    stLENS1_750[0].fEnergy := 5960.000000; stLENS1_750[0].fLow := 85.385702; stLENS1_750[0].fHigh := 10000.000000; 
    stLENS1_750[1].fEnergy := 5972.689818; stLENS1_750[1].fLow := 85.043271; stLENS1_750[1].fHigh := 10000.000000; 
    stLENS1_750[2].fEnergy := 5984.647151; stLENS1_750[2].fLow := 84.702213; stLENS1_750[2].fHigh := 10000.000000; 
    stLENS1_750[3].fEnergy := 5996.628422; stLENS1_750[3].fLow := 84.362523; stLENS1_750[3].fHigh := 10000.000000; 
    stLENS1_750[4].fEnergy := 6008.633680; stLENS1_750[4].fLow := 84.024196; stLENS1_750[4].fHigh := 10000.000000; 
    stLENS1_750[5].fEnergy := 6020.662973; stLENS1_750[5].fLow := 83.687225; stLENS1_750[5].fHigh := 10000.000000; 
    stLENS1_750[6].fEnergy := 6032.716348; stLENS1_750[6].fLow := 83.351606; stLENS1_750[6].fHigh := 10000.000000; 
    stLENS1_750[7].fEnergy := 6044.793854; stLENS1_750[7].fLow := 83.017332; stLENS1_750[7].fHigh := 10000.000000; 
    stLENS1_750[8].fEnergy := 6056.895540; stLENS1_750[8].fLow := 82.684399; stLENS1_750[8].fHigh := 10000.000000; 
    stLENS1_750[9].fEnergy := 6069.021453; stLENS1_750[9].fLow := 82.352801; stLENS1_750[9].fHigh := 10000.000000; 
    stLENS1_750[10].fEnergy := 6081.171642; stLENS1_750[10].fLow := 82.022534; stLENS1_750[10].fHigh := 10000.000000; 
    stLENS1_750[11].fEnergy := 6093.346156; stLENS1_750[11].fLow := 81.693590; stLENS1_750[11].fHigh := 10000.000000; 
    stLENS1_750[12].fEnergy := 6105.545043; stLENS1_750[12].fLow := 81.365966; stLENS1_750[12].fHigh := 10000.000000; 
    stLENS1_750[13].fEnergy := 6117.768352; stLENS1_750[13].fLow := 81.039656; stLENS1_750[13].fHigh := 10000.000000; 
    stLENS1_750[14].fEnergy := 6130.016132; stLENS1_750[14].fLow := 80.714654; stLENS1_750[14].fHigh := 10000.000000; 
    stLENS1_750[15].fEnergy := 6142.288433; stLENS1_750[15].fLow := 80.390956; stLENS1_750[15].fHigh := 10000.000000; 
    stLENS1_750[16].fEnergy := 6154.585303; stLENS1_750[16].fLow := 80.068556; stLENS1_750[16].fHigh := 10000.000000; 
    stLENS1_750[17].fEnergy := 6166.906791; stLENS1_750[17].fLow := 79.747449; stLENS1_750[17].fHigh := 10000.000000; 
    stLENS1_750[18].fEnergy := 6179.252946; stLENS1_750[18].fLow := 79.427629; stLENS1_750[18].fHigh := 10000.000000; 
    stLENS1_750[19].fEnergy := 6191.623819; stLENS1_750[19].fLow := 79.109092; stLENS1_750[19].fHigh := 10000.000000; 
    stLENS1_750[20].fEnergy := 6204.019458; stLENS1_750[20].fLow := 78.791833; stLENS1_750[20].fHigh := 10000.000000; 
    stLENS1_750[21].fEnergy := 6216.439913; stLENS1_750[21].fLow := 78.475846; stLENS1_750[21].fHigh := 10000.000000; 
    stLENS1_750[22].fEnergy := 6228.885234; stLENS1_750[22].fLow := 78.161127; stLENS1_750[22].fHigh := 10000.000000; 
    stLENS1_750[23].fEnergy := 6241.355471; stLENS1_750[23].fLow := 77.847669; stLENS1_750[23].fHigh := 10000.000000; 
    stLENS1_750[24].fEnergy := 6253.850673; stLENS1_750[24].fLow := 77.535468; stLENS1_750[24].fHigh := 10000.000000; 
    stLENS1_750[25].fEnergy := 6266.370890; stLENS1_750[25].fLow := 77.224520; stLENS1_750[25].fHigh := 10000.000000; 
    stLENS1_750[26].fEnergy := 6278.916173; stLENS1_750[26].fLow := 76.914819; stLENS1_750[26].fHigh := 10000.000000; 
    stLENS1_750[27].fEnergy := 6291.486572; stLENS1_750[27].fLow := 76.606359; stLENS1_750[27].fHigh := 10000.000000; 
    stLENS1_750[28].fEnergy := 6304.082136; stLENS1_750[28].fLow := 76.299137; stLENS1_750[28].fHigh := 10000.000000; 
    stLENS1_750[29].fEnergy := 6316.702917; stLENS1_750[29].fLow := 75.993147; stLENS1_750[29].fHigh := 10000.000000; 
    stLENS1_750[30].fEnergy := 6329.348965; stLENS1_750[30].fLow := 75.688384; stLENS1_750[30].fHigh := 10000.000000; 
    stLENS1_750[31].fEnergy := 6342.020330; stLENS1_750[31].fLow := 75.384843; stLENS1_750[31].fHigh := 10000.000000; 
    stLENS1_750[32].fEnergy := 6354.717063; stLENS1_750[32].fLow := 75.082519; stLENS1_750[32].fHigh := 10000.000000; 
    stLENS1_750[33].fEnergy := 6367.439215; stLENS1_750[33].fLow := 74.781408; stLENS1_750[33].fHigh := 10000.000000; 
    stLENS1_750[34].fEnergy := 6380.186837; stLENS1_750[34].fLow := 74.481504; stLENS1_750[34].fHigh := 10000.000000; 
    stLENS1_750[35].fEnergy := 6392.959979; stLENS1_750[35].fLow := 74.182804; stLENS1_750[35].fHigh := 10000.000000; 
    stLENS1_750[36].fEnergy := 6405.758694; stLENS1_750[36].fLow := 73.885301; stLENS1_750[36].fHigh := 10000.000000; 
    stLENS1_750[37].fEnergy := 6418.583031; stLENS1_750[37].fLow := 73.588991; stLENS1_750[37].fHigh := 10000.000000; 
    stLENS1_750[38].fEnergy := 6431.433043; stLENS1_750[38].fLow := 73.293869; stLENS1_750[38].fHigh := 10000.000000; 
    stLENS1_750[39].fEnergy := 6444.308780; stLENS1_750[39].fLow := 72.999932; stLENS1_750[39].fHigh := 10000.000000; 
    stLENS1_750[40].fEnergy := 6457.210295; stLENS1_750[40].fLow := 72.707172; stLENS1_750[40].fHigh := 10000.000000; 
    stLENS1_750[41].fEnergy := 6470.137639; stLENS1_750[41].fLow := 72.415587; stLENS1_750[41].fHigh := 10000.000000; 
    stLENS1_750[42].fEnergy := 6483.090863; stLENS1_750[42].fLow := 72.125172; stLENS1_750[42].fHigh := 10000.000000; 
    stLENS1_750[43].fEnergy := 6496.070019; stLENS1_750[43].fLow := 71.835921; stLENS1_750[43].fHigh := 10000.000000; 
    stLENS1_750[44].fEnergy := 6509.075160; stLENS1_750[44].fLow := 71.547830; stLENS1_750[44].fHigh := 10000.000000; 
    stLENS1_750[45].fEnergy := 6522.106337; stLENS1_750[45].fLow := 71.260894; stLENS1_750[45].fHigh := 10000.000000; 
    stLENS1_750[46].fEnergy := 6535.163603; stLENS1_750[46].fLow := 70.975109; stLENS1_750[46].fHigh := 10000.000000; 
    stLENS1_750[47].fEnergy := 6548.247009; stLENS1_750[47].fLow := 70.690471; stLENS1_750[47].fHigh := 10000.000000; 
    stLENS1_750[48].fEnergy := 6561.356609; stLENS1_750[48].fLow := 70.406973; stLENS1_750[48].fHigh := 10000.000000; 
    stLENS1_750[49].fEnergy := 6574.492453; stLENS1_750[49].fLow := 70.124613; stLENS1_750[49].fHigh := 10000.000000; 
    stLENS1_750[50].fEnergy := 6587.654596; stLENS1_750[50].fLow := 69.843385; stLENS1_750[50].fHigh := 10000.000000; 
    stLENS1_750[51].fEnergy := 6600.843089; stLENS1_750[51].fLow := 69.563285; stLENS1_750[51].fHigh := 10000.000000; 
    stLENS1_750[52].fEnergy := 6614.057986; stLENS1_750[52].fLow := 69.284308; stLENS1_750[52].fHigh := 10000.000000; 
    stLENS1_750[53].fEnergy := 6627.299339; stLENS1_750[53].fLow := 69.006450; stLENS1_750[53].fHigh := 10000.000000; 
    stLENS1_750[54].fEnergy := 6640.567201; stLENS1_750[54].fLow := 68.729707; stLENS1_750[54].fHigh := 10000.000000; 
    stLENS1_750[55].fEnergy := 6653.861625; stLENS1_750[55].fLow := 68.454073; stLENS1_750[55].fHigh := 10000.000000; 
    stLENS1_750[56].fEnergy := 6667.182665; stLENS1_750[56].fLow := 68.179545; stLENS1_750[56].fHigh := 10000.000000; 
    stLENS1_750[57].fEnergy := 6680.530374; stLENS1_750[57].fLow := 67.906117; stLENS1_750[57].fHigh := 10000.000000; 
    stLENS1_750[58].fEnergy := 6693.904804; stLENS1_750[58].fLow := 67.633786; stLENS1_750[58].fHigh := 10000.000000; 
    stLENS1_750[59].fEnergy := 6707.306011; stLENS1_750[59].fLow := 67.362548; stLENS1_750[59].fHigh := 10000.000000; 
    stLENS1_750[60].fEnergy := 6720.734046; stLENS1_750[60].fLow := 67.092397; stLENS1_750[60].fHigh := 10000.000000; 
    stLENS1_750[61].fEnergy := 6734.188965; stLENS1_750[61].fLow := 66.823329; stLENS1_750[61].fHigh := 10000.000000; 
    stLENS1_750[62].fEnergy := 6747.670820; stLENS1_750[62].fLow := 66.555341; stLENS1_750[62].fHigh := 10000.000000; 
    stLENS1_750[63].fEnergy := 6761.179666; stLENS1_750[63].fLow := 66.288427; stLENS1_750[63].fHigh := 10000.000000; 
    stLENS1_750[64].fEnergy := 6774.715557; stLENS1_750[64].fLow := 66.022584; stLENS1_750[64].fHigh := 10000.000000; 
    stLENS1_750[65].fEnergy := 6788.278546; stLENS1_750[65].fLow := 65.757807; stLENS1_750[65].fHigh := 10000.000000; 
    stLENS1_750[66].fEnergy := 6801.868689; stLENS1_750[66].fLow := 65.494091; stLENS1_750[66].fHigh := 10000.000000; 
    stLENS1_750[67].fEnergy := 6815.486039; stLENS1_750[67].fLow := 65.231434; stLENS1_750[67].fHigh := 10000.000000; 
    stLENS1_750[68].fEnergy := 6829.130652; stLENS1_750[68].fLow := 64.969829; stLENS1_750[68].fHigh := 10000.000000; 
    stLENS1_750[69].fEnergy := 6842.802580; stLENS1_750[69].fLow := 64.709274; stLENS1_750[69].fHigh := 10000.000000; 
    stLENS1_750[70].fEnergy := 6856.501880; stLENS1_750[70].fLow := 64.449764; stLENS1_750[70].fHigh := 10000.000000; 
    stLENS1_750[71].fEnergy := 6870.228606; stLENS1_750[71].fLow := 64.191295; stLENS1_750[71].fHigh := 10000.000000; 
    stLENS1_750[72].fEnergy := 6883.982813; stLENS1_750[72].fLow := 63.933862; stLENS1_750[72].fHigh := 10000.000000; 
    stLENS1_750[73].fEnergy := 6897.764556; stLENS1_750[73].fLow := 63.677461; stLENS1_750[73].fHigh := 10000.000000; 
    stLENS1_750[74].fEnergy := 6911.573889; stLENS1_750[74].fLow := 63.422089; stLENS1_750[74].fHigh := 10000.000000; 
    stLENS1_750[75].fEnergy := 6925.410870; stLENS1_750[75].fLow := 63.167741; stLENS1_750[75].fHigh := 10000.000000; 
    stLENS1_750[76].fEnergy := 6939.275551; stLENS1_750[76].fLow := 62.914413; stLENS1_750[76].fHigh := 10000.000000; 
    stLENS1_750[77].fEnergy := 6953.167990; stLENS1_750[77].fLow := 62.662101; stLENS1_750[77].fHigh := 10000.000000; 
    stLENS1_750[78].fEnergy := 6967.088242; stLENS1_750[78].fLow := 62.410800; stLENS1_750[78].fHigh := 10000.000000; 
    stLENS1_750[79].fEnergy := 6981.036362; stLENS1_750[79].fLow := 62.160508; stLENS1_750[79].fHigh := 10000.000000; 
    stLENS1_750[80].fEnergy := 6995.012406; stLENS1_750[80].fLow := 61.911219; stLENS1_750[80].fHigh := 10000.000000; 
    stLENS1_750[81].fEnergy := 7009.016430; stLENS1_750[81].fLow := 61.662930; stLENS1_750[81].fHigh := 10000.000000; 
    stLENS1_750[82].fEnergy := 7023.048490; stLENS1_750[82].fLow := 61.415637; stLENS1_750[82].fHigh := 10000.000000; 
    stLENS1_750[83].fEnergy := 7037.108643; stLENS1_750[83].fLow := 61.169336; stLENS1_750[83].fHigh := 10000.000000; 
    stLENS1_750[84].fEnergy := 7051.196944; stLENS1_750[84].fLow := 60.924022; stLENS1_750[84].fHigh := 10000.000000; 
    stLENS1_750[85].fEnergy := 7065.313449; stLENS1_750[85].fLow := 60.679692; stLENS1_750[85].fHigh := 10000.000000; 
    stLENS1_750[86].fEnergy := 7079.458216; stLENS1_750[86].fLow := 60.436342; stLENS1_750[86].fHigh := 10000.000000; 
    stLENS1_750[87].fEnergy := 7093.631301; stLENS1_750[87].fLow := 60.193968; stLENS1_750[87].fHigh := 10000.000000; 
    stLENS1_750[88].fEnergy := 7107.832760; stLENS1_750[88].fLow := 59.952566; stLENS1_750[88].fHigh := 10000.000000; 
    stLENS1_750[89].fEnergy := 7122.062651; stLENS1_750[89].fLow := 59.712132; stLENS1_750[89].fHigh := 10000.000000; 
    stLENS1_750[90].fEnergy := 7136.321030; stLENS1_750[90].fLow := 59.472663; stLENS1_750[90].fHigh := 10000.000000; 
    stLENS1_750[91].fEnergy := 7150.607954; stLENS1_750[91].fLow := 59.234153; stLENS1_750[91].fHigh := 10000.000000; 
    stLENS1_750[92].fEnergy := 7164.923481; stLENS1_750[92].fLow := 58.996600; stLENS1_750[92].fHigh := 10000.000000; 
    stLENS1_750[93].fEnergy := 7179.267667; stLENS1_750[93].fLow := 58.760000; stLENS1_750[93].fHigh := 10000.000000; 
    stLENS1_750[94].fEnergy := 7193.640571; stLENS1_750[94].fLow := 58.524349; stLENS1_750[94].fHigh := 10000.000000; 
    stLENS1_750[95].fEnergy := 7208.042249; stLENS1_750[95].fLow := 58.289643; stLENS1_750[95].fHigh := 10000.000000; 
    stLENS1_750[96].fEnergy := 7222.472759; stLENS1_750[96].fLow := 58.055878; stLENS1_750[96].fHigh := 10000.000000; 
    stLENS1_750[97].fEnergy := 7236.932159; stLENS1_750[97].fLow := 57.823051; stLENS1_750[97].fHigh := 10000.000000; 
    stLENS1_750[98].fEnergy := 7251.420507; stLENS1_750[98].fLow := 57.591157; stLENS1_750[98].fHigh := 10000.000000; 
    stLENS1_750[99].fEnergy := 7265.937860; stLENS1_750[99].fLow := 57.360193; stLENS1_750[99].fHigh := 10000.000000; 
    stLENS1_750[100].fEnergy := 7280.484278; stLENS1_750[100].fLow := 57.130156; stLENS1_750[100].fHigh := 10000.000000; 
    stLENS1_750[101].fEnergy := 7295.059817; stLENS1_750[101].fLow := 56.901041; stLENS1_750[101].fHigh := 10000.000000; 
    stLENS1_750[102].fEnergy := 7309.664536; stLENS1_750[102].fLow := 56.672845; stLENS1_750[102].fHigh := 10000.000000; 
    stLENS1_750[103].fEnergy := 7324.298495; stLENS1_750[103].fLow := 56.445564; stLENS1_750[103].fHigh := 10000.000000; 
    stLENS1_750[104].fEnergy := 7338.961750; stLENS1_750[104].fLow := 56.187106; stLENS1_750[104].fHigh := 10000.000000; 
    stLENS1_750[105].fEnergy := 7353.654361; stLENS1_750[105].fLow := 55.986290; stLENS1_750[105].fHigh := 10000.000000; 
    stLENS1_750[106].fEnergy := 7368.376387; stLENS1_750[106].fLow := 55.786181; stLENS1_750[106].fHigh := 10000.000000; 
    stLENS1_750[107].fEnergy := 7383.127886; stLENS1_750[107].fLow := 55.586778; stLENS1_750[107].fHigh := 10000.000000; 
    stLENS1_750[108].fEnergy := 7397.908918; stLENS1_750[108].fLow := 55.388078; stLENS1_750[108].fHigh := 10000.000000; 
    stLENS1_750[109].fEnergy := 7412.719542; stLENS1_750[109].fLow := 55.190079; stLENS1_750[109].fHigh := 10000.000000; 
    stLENS1_750[110].fEnergy := 7427.559816; stLENS1_750[110].fLow := 54.992778; stLENS1_750[110].fHigh := 10000.000000; 
    stLENS1_750[111].fEnergy := 7442.429801; stLENS1_750[111].fLow := 54.796173; stLENS1_750[111].fHigh := 10000.000000; 
    stLENS1_750[112].fEnergy := 7457.329555; stLENS1_750[112].fLow := 54.600261; stLENS1_750[112].fHigh := 10000.000000; 
    stLENS1_750[113].fEnergy := 7472.259139; stLENS1_750[113].fLow := 54.405041; stLENS1_750[113].fHigh := 10000.000000; 
    stLENS1_750[114].fEnergy := 7487.218612; stLENS1_750[114].fLow := 54.210508; stLENS1_750[114].fHigh := 10000.000000; 
    stLENS1_750[115].fEnergy := 7502.208033; stLENS1_750[115].fLow := 54.016662; stLENS1_750[115].fHigh := 10000.000000; 
    stLENS1_750[116].fEnergy := 7517.227464; stLENS1_750[116].fLow := 53.823500; stLENS1_750[116].fHigh := 10000.000000; 
    stLENS1_750[117].fEnergy := 7532.276963; stLENS1_750[117].fLow := 53.631019; stLENS1_750[117].fHigh := 10000.000000; 
    stLENS1_750[118].fEnergy := 7547.356592; stLENS1_750[118].fLow := 53.439217; stLENS1_750[118].fHigh := 10000.000000; 
    stLENS1_750[119].fEnergy := 7562.466410; stLENS1_750[119].fLow := 53.248092; stLENS1_750[119].fHigh := 10000.000000; 
    stLENS1_750[120].fEnergy := 7577.606478; stLENS1_750[120].fLow := 53.057641; stLENS1_750[120].fHigh := 10000.000000; 
    stLENS1_750[121].fEnergy := 7592.776856; stLENS1_750[121].fLow := 52.867862; stLENS1_750[121].fHigh := 10000.000000; 
    stLENS1_750[122].fEnergy := 7607.977605; stLENS1_750[122].fLow := 52.678753; stLENS1_750[122].fHigh := 10000.000000; 
    stLENS1_750[123].fEnergy := 7623.208787; stLENS1_750[123].fLow := 52.490311; stLENS1_750[123].fHigh := 10000.000000; 
    stLENS1_750[124].fEnergy := 7638.470461; stLENS1_750[124].fLow := 52.302534; stLENS1_750[124].fHigh := 10000.000000; 
    stLENS1_750[125].fEnergy := 7653.762689; stLENS1_750[125].fLow := 52.115420; stLENS1_750[125].fHigh := 10000.000000; 
    stLENS1_750[126].fEnergy := 7669.085532; stLENS1_750[126].fLow := 51.928966; stLENS1_750[126].fHigh := 10000.000000; 
    stLENS1_750[127].fEnergy := 7684.439051; stLENS1_750[127].fLow := 51.743170; stLENS1_750[127].fHigh := 10000.000000; 
    stLENS1_750[128].fEnergy := 7699.823309; stLENS1_750[128].fLow := 51.558030; stLENS1_750[128].fHigh := 10000.000000; 
    stLENS1_750[129].fEnergy := 7715.238365; stLENS1_750[129].fLow := 51.373544; stLENS1_750[129].fHigh := 10000.000000; 
    stLENS1_750[130].fEnergy := 7730.684283; stLENS1_750[130].fLow := 51.189708; stLENS1_750[130].fHigh := 10000.000000; 
    stLENS1_750[131].fEnergy := 7746.161123; stLENS1_750[131].fLow := 51.006522; stLENS1_750[131].fHigh := 10000.000000; 
    stLENS1_750[132].fEnergy := 7761.668948; stLENS1_750[132].fLow := 50.823982; stLENS1_750[132].fHigh := 10000.000000; 
    stLENS1_750[133].fEnergy := 7777.207819; stLENS1_750[133].fLow := 50.642087; stLENS1_750[133].fHigh := 10000.000000; 
    stLENS1_750[134].fEnergy := 7792.777800; stLENS1_750[134].fLow := 50.460834; stLENS1_750[134].fHigh := 10000.000000; 
    stLENS1_750[135].fEnergy := 7808.378951; stLENS1_750[135].fLow := 50.280221; stLENS1_750[135].fHigh := 10000.000000; 
    stLENS1_750[136].fEnergy := 7824.011336; stLENS1_750[136].fLow := 50.100246; stLENS1_750[136].fHigh := 10000.000000; 
    stLENS1_750[137].fEnergy := 7839.675018; stLENS1_750[137].fLow := 49.920906; stLENS1_750[137].fHigh := 10000.000000; 
    stLENS1_750[138].fEnergy := 7855.370057; stLENS1_750[138].fLow := 49.742199; stLENS1_750[138].fHigh := 10000.000000; 
    stLENS1_750[139].fEnergy := 7871.096519; stLENS1_750[139].fLow := 49.564124; stLENS1_750[139].fHigh := 10000.000000; 
    stLENS1_750[140].fEnergy := 7886.854464; stLENS1_750[140].fLow := 49.386677; stLENS1_750[140].fHigh := 10000.000000; 
    stLENS1_750[141].fEnergy := 7902.643958; stLENS1_750[141].fLow := 49.209858; stLENS1_750[141].fHigh := 10000.000000; 
    stLENS1_750[142].fEnergy := 7918.465061; stLENS1_750[142].fLow := 49.033662; stLENS1_750[142].fHigh := 10000.000000; 
    stLENS1_750[143].fEnergy := 7934.317839; stLENS1_750[143].fLow := 48.858090; stLENS1_750[143].fHigh := 10000.000000; 
    stLENS1_750[144].fEnergy := 7950.202354; stLENS1_750[144].fLow := 48.683137; stLENS1_750[144].fHigh := 10000.000000; 
    stLENS1_750[145].fEnergy := 7966.118670; stLENS1_750[145].fLow := 48.508802; stLENS1_750[145].fHigh := 10000.000000; 
    stLENS1_750[146].fEnergy := 7982.066850; stLENS1_750[146].fLow := 48.335083; stLENS1_750[146].fHigh := 10000.000000; 
    stLENS1_750[147].fEnergy := 7998.046958; stLENS1_750[147].fLow := 48.161978; stLENS1_750[147].fHigh := 10000.000000; 
    stLENS1_750[148].fEnergy := 8014.059059; stLENS1_750[148].fLow := 47.989485; stLENS1_750[148].fHigh := 10000.000000; 
    stLENS1_750[149].fEnergy := 8030.103216; stLENS1_750[149].fLow := 47.817601; stLENS1_750[149].fHigh := 10000.000000; 
    stLENS1_750[150].fEnergy := 8046.179493; stLENS1_750[150].fLow := 47.646324; stLENS1_750[150].fHigh := 10000.000000; 
    stLENS1_750[151].fEnergy := 8062.287955; stLENS1_750[151].fLow := 47.475653; stLENS1_750[151].fHigh := 10000.000000; 
    stLENS1_750[152].fEnergy := 8078.428667; stLENS1_750[152].fLow := 47.305585; stLENS1_750[152].fHigh := 3143.835794; 
    stLENS1_750[153].fEnergy := 8094.601692; stLENS1_750[153].fLow := 47.136117; stLENS1_750[153].fHigh := 2720.776138; 
    stLENS1_750[154].fEnergy := 8110.807095; stLENS1_750[154].fLow := 46.967249; stLENS1_750[154].fHigh := 2354.646769; 
    stLENS1_750[155].fEnergy := 8127.044942; stLENS1_750[155].fLow := 46.798977; stLENS1_750[155].fHigh := 2037.786692; 
    stLENS1_750[156].fEnergy := 8143.315296; stLENS1_750[156].fLow := 46.631301; stLENS1_750[156].fHigh := 1763.565838; 
    stLENS1_750[157].fEnergy := 8159.618224; stLENS1_750[157].fLow := 46.464216; stLENS1_750[157].fHigh := 1526.246332; 
    stLENS1_750[158].fEnergy := 8175.953791; stLENS1_750[158].fLow := 46.297723; stLENS1_750[158].fHigh := 1320.862435; 
    stLENS1_750[159].fEnergy := 8192.322061; stLENS1_750[159].fLow := 46.131818; stLENS1_750[159].fHigh := 1143.116635; 
    stLENS1_750[160].fEnergy := 8208.723101; stLENS1_750[160].fLow := 45.966500; stLENS1_750[160].fHigh := 997.619247; 
    stLENS1_750[161].fEnergy := 8225.156976; stLENS1_750[161].fLow := 45.801766; stLENS1_750[161].fHigh := 966.208437; 
    stLENS1_750[162].fEnergy := 8241.623751; stLENS1_750[162].fLow := 45.637614; stLENS1_750[162].fHigh := 935.786621; 
    stLENS1_750[163].fEnergy := 8258.123493; stLENS1_750[163].fLow := 45.474043; stLENS1_750[163].fHigh := 906.322659; 
    stLENS1_750[164].fEnergy := 8274.656267; stLENS1_750[164].fLow := 45.311050; stLENS1_750[164].fHigh := 877.786393; 
    stLENS1_750[165].fEnergy := 8291.222140; stLENS1_750[165].fLow := 45.148634; stLENS1_750[165].fHigh := 850.148612; 
    stLENS1_750[166].fEnergy := 8307.821178; stLENS1_750[166].fLow := 44.986792; stLENS1_750[166].fHigh := 823.381029; 
    stLENS1_750[167].fEnergy := 8324.453447; stLENS1_750[167].fLow := 44.825522; stLENS1_750[167].fHigh := 797.456244; 
    stLENS1_750[168].fEnergy := 8341.119014; stLENS1_750[168].fLow := 44.664822; stLENS1_750[168].fHigh := 772.347720; 
    stLENS1_750[169].fEnergy := 8357.817945; stLENS1_750[169].fLow := 44.504691; stLENS1_750[169].fHigh := 748.029758; 
    stLENS1_750[170].fEnergy := 8374.550308; stLENS1_750[170].fLow := 44.345127; stLENS1_750[170].fHigh := 724.477465; 
    stLENS1_750[171].fEnergy := 8391.316169; stLENS1_750[171].fLow := 44.186126; stLENS1_750[171].fHigh := 701.666735; 
    stLENS1_750[172].fEnergy := 8408.115595; stLENS1_750[172].fLow := 44.027689; stLENS1_750[172].fHigh := 679.574218; 
    stLENS1_750[173].fEnergy := 8424.948653; stLENS1_750[173].fLow := 43.869811; stLENS1_750[173].fHigh := 658.177300; 
    stLENS1_750[174].fEnergy := 8441.815412; stLENS1_750[174].fLow := 43.712492; stLENS1_750[174].fHigh := 637.454081; 
    stLENS1_750[175].fEnergy := 8458.715938; stLENS1_750[175].fLow := 43.555730; stLENS1_750[175].fHigh := 617.383349; 
    stLENS1_750[176].fEnergy := 8475.650298; stLENS1_750[176].fLow := 43.399523; stLENS1_750[176].fHigh := 597.944559; 
    stLENS1_750[177].fEnergy := 8492.618561; stLENS1_750[177].fLow := 43.243868; stLENS1_750[177].fHigh := 579.117815; 
    stLENS1_750[178].fEnergy := 8509.620795; stLENS1_750[178].fLow := 43.088763; stLENS1_750[178].fHigh := 560.883845; 
    stLENS1_750[179].fEnergy := 8526.657067; stLENS1_750[179].fLow := 42.934208; stLENS1_750[179].fHigh := 543.223985; 
    stLENS1_750[180].fEnergy := 8543.727446; stLENS1_750[180].fLow := 42.780200; stLENS1_750[180].fHigh := 526.120160; 
    stLENS1_750[181].fEnergy := 8560.832000; stLENS1_750[181].fLow := 42.626736; stLENS1_750[181].fHigh := 509.554862; 
    stLENS1_750[182].fEnergy := 8577.970797; stLENS1_750[182].fLow := 42.473816; stLENS1_750[182].fHigh := 493.511135; 
    stLENS1_750[183].fEnergy := 8595.143906; stLENS1_750[183].fLow := 42.321437; stLENS1_750[183].fHigh := 477.972557; 
    stLENS1_750[184].fEnergy := 8612.351395; stLENS1_750[184].fLow := 42.169597; stLENS1_750[184].fHigh := 462.923223; 
    stLENS1_750[185].fEnergy := 8629.593334; stLENS1_750[185].fLow := 42.018295; stLENS1_750[185].fHigh := 448.347729; 
    stLENS1_750[186].fEnergy := 8646.869792; stLENS1_750[186].fLow := 41.867528; stLENS1_750[186].fHigh := 434.231156; 
    stLENS1_750[187].fEnergy := 8664.180837; stLENS1_750[187].fLow := 41.717295; stLENS1_750[187].fHigh := 420.559054; 
    stLENS1_750[188].fEnergy := 8681.526538; stLENS1_750[188].fLow := 41.567594; stLENS1_750[188].fHigh := 407.317428; 
    stLENS1_750[189].fEnergy := 8698.906966; stLENS1_750[189].fLow := 41.418423; stLENS1_750[189].fHigh := 394.492726; 
    stLENS1_750[190].fEnergy := 8716.322189; stLENS1_750[190].fLow := 41.269780; stLENS1_750[190].fHigh := 382.071818; 
    stLENS1_750[191].fEnergy := 8733.772278; stLENS1_750[191].fLow := 41.121663; stLENS1_750[191].fHigh := 370.041993; 
    stLENS1_750[192].fEnergy := 8751.257302; stLENS1_750[192].fLow := 40.974071; stLENS1_750[192].fHigh := 358.390936; 
    stLENS1_750[193].fEnergy := 8768.777330; stLENS1_750[193].fLow := 40.827001; stLENS1_750[193].fHigh := 347.106722; 
    stLENS1_750[194].fEnergy := 8786.332434; stLENS1_750[194].fLow := 40.680452; stLENS1_750[194].fHigh := 336.177800; 
    stLENS1_750[195].fEnergy := 8803.922684; stLENS1_750[195].fLow := 40.534422; stLENS1_750[195].fHigh := 325.592983; 
    stLENS1_750[196].fEnergy := 8821.548149; stLENS1_750[196].fLow := 40.388910; stLENS1_750[196].fHigh := 315.921943; 
    stLENS1_750[197].fEnergy := 8839.208900; stLENS1_750[197].fLow := 40.243912; stLENS1_750[197].fHigh := 312.455190; 
    stLENS1_750[198].fEnergy := 8856.905008; stLENS1_750[198].fLow := 40.099428; stLENS1_750[198].fHigh := 309.026479; 
    stLENS1_750[199].fEnergy := 8874.636543; stLENS1_750[199].fLow := 39.955456; stLENS1_750[199].fHigh := 305.635394; 
    stLENS1_750[200].fEnergy := 8892.403578; stLENS1_750[200].fLow := 39.811994; stLENS1_750[200].fHigh := 302.281520; 
    stLENS1_750[201].fEnergy := 8910.206181; stLENS1_750[201].fLow := 39.669040; stLENS1_750[201].fHigh := 298.964450; 
    stLENS1_750[202].fEnergy := 8928.044426; stLENS1_750[202].fLow := 39.526593; stLENS1_750[202].fHigh := 295.683779; 
    stLENS1_750[203].fEnergy := 8945.918383; stLENS1_750[203].fLow := 39.384650; stLENS1_750[203].fHigh := 292.439109; 
    stLENS1_750[204].fEnergy := 8963.828123; stLENS1_750[204].fLow := 39.243210; stLENS1_750[204].fHigh := 289.230044; 
    stLENS1_750[205].fEnergy := 8981.773719; stLENS1_750[205].fLow := 39.102272; stLENS1_750[205].fHigh := 286.056193; 
    stLENS1_750[206].fEnergy := 8999.755242; stLENS1_750[206].fLow := 38.961832; stLENS1_750[206].fHigh := 282.917171; 
    stLENS1_750[207].fEnergy := 9017.772764; stLENS1_750[207].fLow := 38.821891; stLENS1_750[207].fHigh := 279.812594; 
    stLENS1_750[208].fEnergy := 9035.826357; stLENS1_750[208].fLow := 38.682445; stLENS1_750[208].fHigh := 276.742086; 
    stLENS1_750[209].fEnergy := 9053.916094; stLENS1_750[209].fLow := 38.543493; stLENS1_750[209].fHigh := 273.705271; 
    stLENS1_750[210].fEnergy := 9072.042046; stLENS1_750[210].fLow := 38.405034; stLENS1_750[210].fHigh := 270.701781; 
    stLENS1_750[211].fEnergy := 9090.204286; stLENS1_750[211].fLow := 38.267065; stLENS1_750[211].fHigh := 267.731249; 
    stLENS1_750[212].fEnergy := 9108.402887; stLENS1_750[212].fLow := 38.129586; stLENS1_750[212].fHigh := 264.793314; 
    stLENS1_750[213].fEnergy := 9126.637922; stLENS1_750[213].fLow := 37.992594; stLENS1_750[213].fHigh := 261.887619; 
    stLENS1_750[214].fEnergy := 9144.909463; stLENS1_750[214].fLow := 37.856087; stLENS1_750[214].fHigh := 259.013809; 
    stLENS1_750[215].fEnergy := 9163.217584; stLENS1_750[215].fLow := 37.720065; stLENS1_750[215].fHigh := 256.171535; 
    stLENS1_750[216].fEnergy := 9181.562358; stLENS1_750[216].fLow := 37.584524; stLENS1_750[216].fHigh := 253.360450; 
    stLENS1_750[217].fEnergy := 9199.943858; stLENS1_750[217].fLow := 37.449464; stLENS1_750[217].fHigh := 250.580213; 
    stLENS1_750[218].fEnergy := 9218.362158; stLENS1_750[218].fLow := 37.314883; stLENS1_750[218].fHigh := 247.830484; 
    stLENS1_750[219].fEnergy := 9236.817331; stLENS1_750[219].fLow := 37.180779; stLENS1_750[219].fHigh := 245.110929; 
    stLENS1_750[220].fEnergy := 9255.309452; stLENS1_750[220].fLow := 37.047151; stLENS1_750[220].fHigh := 242.421218; 
    stLENS1_750[221].fEnergy := 9273.838594; stLENS1_750[221].fLow := 36.913996; stLENS1_750[221].fHigh := 239.761021; 
    stLENS1_750[222].fEnergy := 9292.404831; stLENS1_750[222].fLow := 36.781314; stLENS1_750[222].fHigh := 237.130016; 
    stLENS1_750[223].fEnergy := 9311.008238; stLENS1_750[223].fLow := 36.649102; stLENS1_750[223].fHigh := 234.527883; 
    stLENS1_750[224].fEnergy := 9329.648889; stLENS1_750[224].fLow := 36.517359; stLENS1_750[224].fHigh := 231.954303; 
    stLENS1_750[225].fEnergy := 9348.326858; stLENS1_750[225].fLow := 36.386083; stLENS1_750[225].fHigh := 229.408965; 
    stLENS1_750[226].fEnergy := 9367.042221; stLENS1_750[226].fLow := 36.255273; stLENS1_750[226].fHigh := 226.891558; 
    stLENS1_750[227].fEnergy := 9385.795052; stLENS1_750[227].fLow := 36.124927; stLENS1_750[227].fHigh := 224.401776; 
    stLENS1_750[228].fEnergy := 9404.585426; stLENS1_750[228].fLow := 35.995043; stLENS1_750[228].fHigh := 221.939315; 
    stLENS1_750[229].fEnergy := 9423.413419; stLENS1_750[229].fLow := 35.865620; stLENS1_750[229].fHigh := 219.503875; 
    stLENS1_750[230].fEnergy := 9442.279105; stLENS1_750[230].fLow := 35.736656; stLENS1_750[230].fHigh := 217.095161; 
    stLENS1_750[231].fEnergy := 9461.182561; stLENS1_750[231].fLow := 35.608149; stLENS1_750[231].fHigh := 214.712879; 
    stLENS1_750[232].fEnergy := 9480.123861; stLENS1_750[232].fLow := 35.480099; stLENS1_750[232].fHigh := 212.356739; 
    stLENS1_750[233].fEnergy := 9499.103081; stLENS1_750[233].fLow := 35.352503; stLENS1_750[233].fHigh := 210.026453; 
    stLENS1_750[234].fEnergy := 9518.120298; stLENS1_750[234].fLow := 35.225359; stLENS1_750[234].fHigh := 207.721739; 
    stLENS1_750[235].fEnergy := 9537.175588; stLENS1_750[235].fLow := 35.098667; stLENS1_750[235].fHigh := 205.442316; 
    stLENS1_750[236].fEnergy := 9556.269026; stLENS1_750[236].fLow := 34.972424; stLENS1_750[236].fHigh := 203.187905; 
    stLENS1_750[237].fEnergy := 9575.400690; stLENS1_750[237].fLow := 34.846629; stLENS1_750[237].fHigh := 200.958233; 
    stLENS1_750[238].fEnergy := 9594.570654; stLENS1_750[238].fLow := 34.721281; stLENS1_750[238].fHigh := 198.753029; 
    stLENS1_750[239].fEnergy := 9613.778998; stLENS1_750[239].fLow := 34.596378; stLENS1_750[239].fHigh := 196.572023; 
    stLENS1_750[240].fEnergy := 9633.025796; stLENS1_750[240].fLow := 34.471917; stLENS1_750[240].fHigh := 194.414950; 
    stLENS1_750[241].fEnergy := 9652.311127; stLENS1_750[241].fLow := 34.347899; stLENS1_750[241].fHigh := 192.281548; 
    stLENS1_750[242].fEnergy := 9671.635066; stLENS1_750[242].fLow := 34.224321; stLENS1_750[242].fHigh := 190.171557; 
    stLENS1_750[243].fEnergy := 9690.997693; stLENS1_750[243].fLow := 34.101182; stLENS1_750[243].fHigh := 188.084719; 
    stLENS1_750[244].fEnergy := 9710.399083; stLENS1_750[244].fLow := 33.978479; stLENS1_750[244].fHigh := 186.020782; 
    stLENS1_750[245].fEnergy := 9729.839315; stLENS1_750[245].fLow := 33.856213; stLENS1_750[245].fHigh := 183.979493; 
    stLENS1_750[246].fEnergy := 9749.318466; stLENS1_750[246].fLow := 33.734380; stLENS1_750[246].fHigh := 181.960603; 
    stLENS1_750[247].fEnergy := 9768.836615; stLENS1_750[247].fLow := 33.612980; stLENS1_750[247].fHigh := 179.963868; 
    stLENS1_750[248].fEnergy := 9788.393839; stLENS1_750[248].fLow := 33.492011; stLENS1_750[248].fHigh := 177.926632; 
    stLENS1_750[249].fEnergy := 9807.990216; stLENS1_750[249].fLow := 33.371471; stLENS1_750[249].fHigh := 176.728069; 
    stLENS1_750[250].fEnergy := 9827.625826; stLENS1_750[250].fLow := 33.251360; stLENS1_750[250].fHigh := 175.537579; 
    stLENS1_750[251].fEnergy := 9847.300746; stLENS1_750[251].fLow := 33.131675; stLENS1_750[251].fHigh := 174.355109; 
    stLENS1_750[252].fEnergy := 9867.015055; stLENS1_750[252].fLow := 33.012415; stLENS1_750[252].fHigh := 173.180604; 
    stLENS1_750[253].fEnergy := 9886.768832; stLENS1_750[253].fLow := 32.893579; stLENS1_750[253].fHigh := 172.014011; 
    stLENS1_750[254].fEnergy := 9906.562157; stLENS1_750[254].fLow := 32.775165; stLENS1_750[254].fHigh := 170.855277; 
    stLENS1_750[255].fEnergy := 9926.395107; stLENS1_750[255].fLow := 32.657171; stLENS1_750[255].fHigh := 169.704348; 
    stLENS1_750[256].fEnergy := 9946.267764; stLENS1_750[256].fLow := 32.539597; stLENS1_750[256].fHigh := 168.561172; 
    stLENS1_750[257].fEnergy := 9966.180205; stLENS1_750[257].fLow := 32.422440; stLENS1_750[257].fHigh := 167.425697; 
    stLENS1_750[258].fEnergy := 9986.132511; stLENS1_750[258].fLow := 32.305699; stLENS1_750[258].fHigh := 166.297870; 
    stLENS1_750[259].fEnergy := 10006.124762; stLENS1_750[259].fLow := 32.189373; stLENS1_750[259].fHigh := 165.177641; 
    stLENS1_750[260].fEnergy := 10026.157037; stLENS1_750[260].fLow := 32.073461; stLENS1_750[260].fHigh := 164.064959; 
    stLENS1_750[261].fEnergy := 10046.229416; stLENS1_750[261].fLow := 31.957960; stLENS1_750[261].fHigh := 162.959771; 
    stLENS1_750[262].fEnergy := 10066.341981; stLENS1_750[262].fLow := 31.842870; stLENS1_750[262].fHigh := 161.862028; 
    stLENS1_750[263].fEnergy := 10086.494811; stLENS1_750[263].fLow := 31.728188; stLENS1_750[263].fHigh := 160.771681; 
    stLENS1_750[264].fEnergy := 10106.687987; stLENS1_750[264].fLow := 31.613914; stLENS1_750[264].fHigh := 159.688678; 
    stLENS1_750[265].fEnergy := 10126.921590; stLENS1_750[265].fLow := 31.500046; stLENS1_750[265].fHigh := 158.612970; 
    stLENS1_750[266].fEnergy := 10147.195701; stLENS1_750[266].fLow := 31.386583; stLENS1_750[266].fHigh := 157.544509; 
    stLENS1_750[267].fEnergy := 10167.510400; stLENS1_750[267].fLow := 31.273523; stLENS1_750[267].fHigh := 156.483245; 
    stLENS1_750[268].fEnergy := 10187.865769; stLENS1_750[268].fLow := 31.160865; stLENS1_750[268].fHigh := 155.429130; 
    stLENS1_750[269].fEnergy := 10208.261890; stLENS1_750[269].fLow := 31.048607; stLENS1_750[269].fHigh := 154.382116; 
    stLENS1_750[270].fEnergy := 10228.698844; stLENS1_750[270].fLow := 30.936749; stLENS1_750[270].fHigh := 153.342155; 
    stLENS1_750[271].fEnergy := 10249.176713; stLENS1_750[271].fLow := 30.825288; stLENS1_750[271].fHigh := 152.309199; 
    stLENS1_750[272].fEnergy := 10269.695578; stLENS1_750[272].fLow := 30.714223; stLENS1_750[272].fHigh := 151.283202; 
    stLENS1_750[273].fEnergy := 10290.255523; stLENS1_750[273].fLow := 30.603553; stLENS1_750[273].fHigh := 150.264116; 
    stLENS1_750[274].fEnergy := 10310.856628; stLENS1_750[274].fLow := 30.493277; stLENS1_750[274].fHigh := 149.251895; 
    stLENS1_750[275].fEnergy := 10331.498977; stLENS1_750[275].fLow := 30.383392; stLENS1_750[275].fHigh := 148.246492; 
    stLENS1_750[276].fEnergy := 10352.182651; stLENS1_750[276].fLow := 30.273899; stLENS1_750[276].fHigh := 147.247862; 
    stLENS1_750[277].fEnergy := 10372.907735; stLENS1_750[277].fLow := 30.164794; stLENS1_750[277].fHigh := 146.255959; 
    stLENS1_750[278].fEnergy := 10393.674310; stLENS1_750[278].fLow := 30.056078; stLENS1_750[278].fHigh := 145.270738; 
    stLENS1_750[279].fEnergy := 10414.482460; stLENS1_750[279].fLow := 29.947748; stLENS1_750[279].fHigh := 144.292154; 
    stLENS1_750[280].fEnergy := 10435.332268; stLENS1_750[280].fLow := 29.839803; stLENS1_750[280].fHigh := 143.320162; 
    stLENS1_750[281].fEnergy := 10456.223817; stLENS1_750[281].fLow := 29.732243; stLENS1_750[281].fHigh := 142.354717; 
    stLENS1_750[282].fEnergy := 10477.157191; stLENS1_750[282].fLow := 29.625065; stLENS1_750[282].fHigh := 141.395776; 
    stLENS1_750[283].fEnergy := 10498.132473; stLENS1_750[283].fLow := 29.518268; stLENS1_750[283].fHigh := 140.443294; 
    stLENS1_750[284].fEnergy := 10519.149749; stLENS1_750[284].fLow := 29.411851; stLENS1_750[284].fHigh := 139.497229; 
    stLENS1_750[285].fEnergy := 10540.209100; stLENS1_750[285].fLow := 29.305812; stLENS1_750[285].fHigh := 138.557537; 
    stLENS1_750[286].fEnergy := 10561.310613; stLENS1_750[286].fLow := 29.200151; stLENS1_750[286].fHigh := 137.624174; 
    stLENS1_750[287].fEnergy := 10582.454371; stLENS1_750[287].fLow := 29.094866; stLENS1_750[287].fHigh := 136.697100; 
    stLENS1_750[288].fEnergy := 10603.640459; stLENS1_750[288].fLow := 28.989955; stLENS1_750[288].fHigh := 135.776270; 
    stLENS1_750[289].fEnergy := 10624.868961; stLENS1_750[289].fLow := 28.885418; stLENS1_750[289].fHigh := 134.861643; 
    stLENS1_750[290].fEnergy := 10646.139963; stLENS1_750[290].fLow := 28.781252; stLENS1_750[290].fHigh := 133.953177; 
    stLENS1_750[291].fEnergy := 10667.453549; stLENS1_750[291].fLow := 28.677457; stLENS1_750[291].fHigh := 133.050831; 
    stLENS1_750[292].fEnergy := 10688.809806; stLENS1_750[292].fLow := 28.574031; stLENS1_750[292].fHigh := 132.154563; 
    stLENS1_750[293].fEnergy := 10710.208817; stLENS1_750[293].fLow := 28.470974; stLENS1_750[293].fHigh := 131.264333; 
    stLENS1_750[294].fEnergy := 10731.650669; stLENS1_750[294].fLow := 28.368283; stLENS1_750[294].fHigh := 130.380100; 
    stLENS1_750[295].fEnergy := 10753.135448; stLENS1_750[295].fLow := 28.265958; stLENS1_750[295].fHigh := 129.501823; 
    stLENS1_750[296].fEnergy := 10774.663240; stLENS1_750[296].fLow := 28.163997; stLENS1_750[296].fHigh := 128.629463; 
    stLENS1_750[297].fEnergy := 10796.234130; stLENS1_750[297].fLow := 28.062399; stLENS1_750[297].fHigh := 127.762979; 
    stLENS1_750[298].fEnergy := 10817.848205; stLENS1_750[298].fLow := 27.961162; stLENS1_750[298].fHigh := 126.902331; 
    stLENS1_750[299].fEnergy := 10839.505552; stLENS1_750[299].fLow := 27.860286; stLENS1_750[299].fHigh := 126.047482; 
    stLENS1_750[300].fEnergy := 10861.206256; stLENS1_750[300].fLow := 27.759769; stLENS1_750[300].fHigh := 125.198391; 
    stLENS1_750[301].fEnergy := 10882.950406; stLENS1_750[301].fLow := 27.659609; stLENS1_750[301].fHigh := 124.355019; 
    stLENS1_750[302].fEnergy := 10904.738087; stLENS1_750[302].fLow := 27.559807; stLENS1_750[302].fHigh := 123.517329; 
    stLENS1_750[303].fEnergy := 10926.569387; stLENS1_750[303].fLow := 27.460359; stLENS1_750[303].fHigh := 122.685282; 
    stLENS1_750[304].fEnergy := 10948.444394; stLENS1_750[304].fLow := 27.361266; stLENS1_750[304].fHigh := 121.858840; 
    stLENS1_750[305].fEnergy := 10970.363194; stLENS1_750[305].fLow := 27.262526; stLENS1_750[305].fHigh := 121.037964; 
    stLENS1_750[306].fEnergy := 10992.325876; stLENS1_750[306].fLow := 27.164137; stLENS1_750[306].fHigh := 120.222619; 
    stLENS1_750[307].fEnergy := 11014.332527; stLENS1_750[307].fLow := 27.066098; stLENS1_750[307].fHigh := 119.412766; 
    stLENS1_750[308].fEnergy := 11036.383235; stLENS1_750[308].fLow := 26.968409; stLENS1_750[308].fHigh := 118.608368; 
    stLENS1_750[309].fEnergy := 11058.478089; stLENS1_750[309].fLow := 26.871068; stLENS1_750[309].fHigh := 117.809389; 
    stLENS1_750[310].fEnergy := 11080.617177; stLENS1_750[310].fLow := 26.774073; stLENS1_750[310].fHigh := 117.015792; 
    stLENS1_750[311].fEnergy := 11102.800587; stLENS1_750[311].fLow := 26.677424; stLENS1_750[311].fHigh := 116.227541; 
    stLENS1_750[312].fEnergy := 11125.028409; stLENS1_750[312].fLow := 26.581119; stLENS1_750[312].fHigh := 115.444599; 
    stLENS1_750[313].fEnergy := 11147.300731; stLENS1_750[313].fLow := 26.485157; stLENS1_750[313].fHigh := 114.666932; 
    stLENS1_750[314].fEnergy := 11169.617642; stLENS1_750[314].fLow := 26.389537; stLENS1_750[314].fHigh := 113.894504; 
    stLENS1_750[315].fEnergy := 11191.979231; stLENS1_750[315].fLow := 26.294257; stLENS1_750[315].fHigh := 113.127278; 
    stLENS1_750[316].fEnergy := 11214.385588; stLENS1_750[316].fLow := 26.199317; stLENS1_750[316].fHigh := 112.365221; 
    stLENS1_750[317].fEnergy := 11236.836803; stLENS1_750[317].fLow := 26.104715; stLENS1_750[317].fHigh := 111.608298; 
    stLENS1_750[318].fEnergy := 11259.332966; stLENS1_750[318].fLow := 26.010451; stLENS1_750[318].fHigh := 110.856473; 
    stLENS1_750[319].fEnergy := 11281.874165; stLENS1_750[319].fLow := 25.916522; stLENS1_750[319].fHigh := 110.109713; 
    stLENS1_750[320].fEnergy := 11304.460492; stLENS1_750[320].fLow := 25.822928; stLENS1_750[320].fHigh := 109.367983; 
    stLENS1_750[321].fEnergy := 11327.092037; stLENS1_750[321].fLow := 25.729667; stLENS1_750[321].fHigh := 108.631250; 
    stLENS1_750[322].fEnergy := 11349.768891; stLENS1_750[322].fLow := 25.636739; stLENS1_750[322].fHigh := 107.899479; 
    stLENS1_750[323].fEnergy := 11372.491143; stLENS1_750[323].fLow := 25.544142; stLENS1_750[323].fHigh := 107.172638; 
    stLENS1_750[324].fEnergy := 11395.258886; stLENS1_750[324].fLow := 25.451875; stLENS1_750[324].fHigh := 106.450693; 
    stLENS1_750[325].fEnergy := 11418.072209; stLENS1_750[325].fLow := 25.359937; stLENS1_750[325].fHigh := 105.733612; 
    stLENS1_750[326].fEnergy := 11440.931205; stLENS1_750[326].fLow := 25.268326; stLENS1_750[326].fHigh := 105.021361; 
    stLENS1_750[327].fEnergy := 11463.835964; stLENS1_750[327].fLow := 25.177042; stLENS1_750[327].fHigh := 104.313907; 
    stLENS1_750[328].fEnergy := 11486.786579; stLENS1_750[328].fLow := 25.086084; stLENS1_750[328].fHigh := 103.611220; 
    stLENS1_750[329].fEnergy := 11509.783141; stLENS1_750[329].fLow := 24.995449; stLENS1_750[329].fHigh := 102.913266; 
    stLENS1_750[330].fEnergy := 11532.825743; stLENS1_750[330].fLow := 24.905138; stLENS1_750[330].fHigh := 102.220013; 
    stLENS1_750[331].fEnergy := 11555.914475; stLENS1_750[331].fLow := 24.815149; stLENS1_750[331].fHigh := 101.531430; 
    stLENS1_750[332].fEnergy := 11579.049431; stLENS1_750[332].fLow := 24.725481; stLENS1_750[332].fHigh := 100.847486; 
    stLENS1_750[333].fEnergy := 11602.230704; stLENS1_750[333].fLow := 24.636132; stLENS1_750[333].fHigh := 100.133379; 
    stLENS1_750[334].fEnergy := 11625.458385; stLENS1_750[334].fLow := 24.547102; stLENS1_750[334].fHigh := 99.597866; 
    stLENS1_750[335].fEnergy := 11648.732568; stLENS1_750[335].fLow := 24.458390; stLENS1_750[335].fHigh := 99.065216; 
    stLENS1_750[336].fEnergy := 11672.053346; stLENS1_750[336].fLow := 24.369993; stLENS1_750[336].fHigh := 98.535415; 
    stLENS1_750[337].fEnergy := 11695.420813; stLENS1_750[337].fLow := 24.281913; stLENS1_750[337].fHigh := 98.008448; 
    stLENS1_750[338].fEnergy := 11718.835061; stLENS1_750[338].fLow := 24.194146; stLENS1_750[338].fHigh := 97.484299; 
    stLENS1_750[339].fEnergy := 11742.296184; stLENS1_750[339].fLow := 24.106692; stLENS1_750[339].fHigh := 96.962952; 
    stLENS1_750[340].fEnergy := 11765.804277; stLENS1_750[340].fLow := 24.019550; stLENS1_750[340].fHigh := 96.444394; 
    stLENS1_750[341].fEnergy := 11789.359433; stLENS1_750[341].fLow := 23.932719; stLENS1_750[341].fHigh := 95.928610; 
    stLENS1_750[342].fEnergy := 11812.961746; stLENS1_750[342].fLow := 23.846198; stLENS1_750[342].fHigh := 95.415583; 
    stLENS1_750[343].fEnergy := 11836.611311; stLENS1_750[343].fLow := 23.759985; stLENS1_750[343].fHigh := 94.905301; 
    stLENS1_750[344].fEnergy := 11860.308223; stLENS1_750[344].fLow := 23.674080; stLENS1_750[344].fHigh := 94.397747; 
    stLENS1_750[345].fEnergy := 11884.052576; stLENS1_750[345].fLow := 23.588482; stLENS1_750[345].fHigh := 93.892908; 
    stLENS1_750[346].fEnergy := 11907.844465; stLENS1_750[346].fLow := 23.503189; stLENS1_750[346].fHigh := 93.390768; 
    stLENS1_750[347].fEnergy := 11931.683985; stLENS1_750[347].fLow := 23.418200; stLENS1_750[347].fHigh := 92.891314; 
    stLENS1_750[348].fEnergy := 11955.571233; stLENS1_750[348].fLow := 23.333514; stLENS1_750[348].fHigh := 92.394531; 
    stLENS1_750[349].fEnergy := 11979.506302; stLENS1_750[349].fLow := 23.249131; stLENS1_750[349].fHigh := 91.900405; 
    stLENS1_750[350].fEnergy := 12003.489290; stLENS1_750[350].fLow := 23.165049; stLENS1_750[350].fHigh := 91.408922; 
    stLENS1_750[351].fEnergy := 12027.520291; stLENS1_750[351].fLow := 23.081267; stLENS1_750[351].fHigh := 90.920067; 
    stLENS1_750[352].fEnergy := 12051.599403; stLENS1_750[352].fLow := 22.997784; stLENS1_750[352].fHigh := 90.433826; 
    stLENS1_750[353].fEnergy := 12075.726721; stLENS1_750[353].fLow := 22.914599; stLENS1_750[353].fHigh := 89.950186; 
    stLENS1_750[354].fEnergy := 12099.902342; stLENS1_750[354].fLow := 22.831710; stLENS1_750[354].fHigh := 89.469132; 
    stLENS1_750[355].fEnergy := 12124.126363; stLENS1_750[355].fLow := 22.749118; stLENS1_750[355].fHigh := 88.990651; 
    stLENS1_750[356].fEnergy := 12148.398880; stLENS1_750[356].fLow := 22.666820; stLENS1_750[356].fHigh := 88.514729; 
    stLENS1_750[357].fEnergy := 12172.719991; stLENS1_750[357].fLow := 22.584817; stLENS1_750[357].fHigh := 88.041352; 
    stLENS1_750[358].fEnergy := 12197.089792; stLENS1_750[358].fLow := 22.503106; stLENS1_750[358].fHigh := 87.570507; 
    stLENS1_750[359].fEnergy := 12221.508382; stLENS1_750[359].fLow := 22.421686; stLENS1_750[359].fHigh := 87.102180; 
    stLENS1_750[360].fEnergy := 12245.975858; stLENS1_750[360].fLow := 22.340558; stLENS1_750[360].fHigh := 86.636357; 
    stLENS1_750[361].fEnergy := 12270.492318; stLENS1_750[361].fLow := 22.259719; stLENS1_750[361].fHigh := 86.173026; 
    stLENS1_750[362].fEnergy := 12295.057860; stLENS1_750[362].fLow := 22.179169; stLENS1_750[362].fHigh := 85.712172; 
    stLENS1_750[363].fEnergy := 12319.672583; stLENS1_750[363].fLow := 22.098906; stLENS1_750[363].fHigh := 85.253784; 
    stLENS1_750[364].fEnergy := 12344.336584; stLENS1_750[364].fLow := 22.018930; stLENS1_750[364].fHigh := 84.797846; 
    stLENS1_750[365].fEnergy := 12369.049962; stLENS1_750[365].fLow := 21.939240; stLENS1_750[365].fHigh := 84.344347; 
    stLENS1_750[366].fEnergy := 12393.812816; stLENS1_750[366].fLow := 21.859834; stLENS1_750[366].fHigh := 83.893274; 
    stLENS1_750[367].fEnergy := 12418.625246; stLENS1_750[367].fLow := 21.780712; stLENS1_750[367].fHigh := 83.444612; 
    stLENS1_750[368].fEnergy := 12443.487350; stLENS1_750[368].fLow := 21.701872; stLENS1_750[368].fHigh := 82.998350; 
    stLENS1_750[369].fEnergy := 12468.399229; stLENS1_750[369].fLow := 21.623314; stLENS1_750[369].fHigh := 82.554475; 
    stLENS1_750[370].fEnergy := 12493.360981; stLENS1_750[370].fLow := 21.545037; stLENS1_750[370].fHigh := 82.112974; 
    stLENS1_750[371].fEnergy := 12518.372706; stLENS1_750[371].fLow := 21.467039; stLENS1_750[371].fHigh := 81.673833; 
    stLENS1_750[372].fEnergy := 12543.434505; stLENS1_750[372].fLow := 21.389320; stLENS1_750[372].fHigh := 81.237042; 
    stLENS1_750[373].fEnergy := 12568.546477; stLENS1_750[373].fLow := 21.311879; stLENS1_750[373].fHigh := 80.802586; 
    stLENS1_750[374].fEnergy := 12593.708724; stLENS1_750[374].fLow := 21.234714; stLENS1_750[374].fHigh := 80.370453; 
    stLENS1_750[375].fEnergy := 12618.921346; stLENS1_750[375].fLow := 21.157825; stLENS1_750[375].fHigh := 79.940632; 
    stLENS1_750[376].fEnergy := 12644.184443; stLENS1_750[376].fLow := 21.081211; stLENS1_750[376].fHigh := 79.513110; 
    stLENS1_750[377].fEnergy := 12669.498117; stLENS1_750[377].fLow := 21.004870; stLENS1_750[377].fHigh := 79.087873; 
    stLENS1_750[378].fEnergy := 12694.862470; stLENS1_750[378].fLow := 20.928802; stLENS1_750[378].fHigh := 78.664911; 
    stLENS1_750[379].fEnergy := 12720.277601; stLENS1_750[379].fLow := 20.853007; stLENS1_750[379].fHigh := 78.244211; 
    stLENS1_750[380].fEnergy := 12745.743614; stLENS1_750[380].fLow := 20.777482; stLENS1_750[380].fHigh := 77.825761; 
    stLENS1_750[381].fEnergy := 12771.260610; stLENS1_750[381].fLow := 20.702227; stLENS1_750[381].fHigh := 77.409549; 
    stLENS1_750[382].fEnergy := 12796.828690; stLENS1_750[382].fLow := 20.627240; stLENS1_750[382].fHigh := 76.995562; 
    stLENS1_750[383].fEnergy := 12822.447958; stLENS1_750[383].fLow := 20.552522; stLENS1_750[383].fHigh := 76.583790; 
    stLENS1_750[384].fEnergy := 12848.118516; stLENS1_750[384].fLow := 20.478071; stLENS1_750[384].fHigh := 76.174220; 
    stLENS1_750[385].fEnergy := 12873.840467; stLENS1_750[385].fLow := 20.403887; stLENS1_750[385].fHigh := 75.766840; 
    stLENS1_750[386].fEnergy := 12899.613913; stLENS1_750[386].fLow := 20.329967; stLENS1_750[386].fHigh := 75.361639; 
    stLENS1_750[387].fEnergy := 12925.438957; stLENS1_750[387].fLow := 20.256312; stLENS1_750[387].fHigh := 74.958605; 
    stLENS1_750[388].fEnergy := 12951.315703; stLENS1_750[388].fLow := 20.182920; stLENS1_750[388].fHigh := 74.557726; 
    stLENS1_750[389].fEnergy := 12977.244254; stLENS1_750[389].fLow := 20.109790; stLENS1_750[389].fHigh := 74.158991; 
    stLENS1_750[390].fEnergy := 13003.224714; stLENS1_750[390].fLow := 20.036922; stLENS1_750[390].fHigh := 73.762389; 
    stLENS1_750[391].fEnergy := 13029.257188; stLENS1_750[391].fLow := 19.964315; stLENS1_750[391].fHigh := 73.367907; 
    stLENS1_750[392].fEnergy := 13055.341778; stLENS1_750[392].fLow := 19.891967; stLENS1_750[392].fHigh := 72.975536; 
    stLENS1_750[393].fEnergy := 13081.478590; stLENS1_750[393].fLow := 19.819877; stLENS1_750[393].fHigh := 72.585262; 
    stLENS1_750[394].fEnergy := 13107.667727; stLENS1_750[394].fLow := 19.748046; stLENS1_750[394].fHigh := 72.197076; 
    stLENS1_750[395].fEnergy := 13133.909296; stLENS1_750[395].fLow := 19.676472; stLENS1_750[395].fHigh := 71.810966; 
    stLENS1_750[396].fEnergy := 13160.203399; stLENS1_750[396].fLow := 19.605153; stLENS1_750[396].fHigh := 71.426921; 
    stLENS1_750[397].fEnergy := 13186.550144; stLENS1_750[397].fLow := 19.534090; stLENS1_750[397].fHigh := 71.044930; 
    stLENS1_750[398].fEnergy := 13212.949635; stLENS1_750[398].fLow := 19.463281; stLENS1_750[398].fHigh := 70.664982; 
    stLENS1_750[399].fEnergy := 13239.401978; stLENS1_750[399].fLow := 19.392725; stLENS1_750[399].fHigh := 70.287065; 
    stLENS1_750[400].fEnergy := 13265.907278; stLENS1_750[400].fLow := 19.322421; stLENS1_750[400].fHigh := 69.911170; 
    stLENS1_750[401].fEnergy := 13292.465642; stLENS1_750[401].fLow := 19.252370; stLENS1_750[401].fHigh := 69.537285; 
    stLENS1_750[402].fEnergy := 13319.077176; stLENS1_750[402].fLow := 19.182568; stLENS1_750[402].fHigh := 69.165399; 
    stLENS1_750[403].fEnergy := 13345.741987; stLENS1_750[403].fLow := 19.113017; stLENS1_750[403].fHigh := 68.795503; 
    stLENS1_750[404].fEnergy := 13372.460180; stLENS1_750[404].fLow := 19.043714; stLENS1_750[404].fHigh := 68.427584; 
    stLENS1_750[405].fEnergy := 13399.231863; stLENS1_750[405].fLow := 18.974659; stLENS1_750[405].fHigh := 68.061633; 
    stLENS1_750[406].fEnergy := 13426.057143; stLENS1_750[406].fLow := 18.905852; stLENS1_750[406].fHigh := 67.697640; 
    stLENS1_750[407].fEnergy := 13452.936127; stLENS1_750[407].fLow := 18.837290; stLENS1_750[407].fHigh := 67.335593; 
    stLENS1_750[408].fEnergy := 13479.868924; stLENS1_750[408].fLow := 18.768974; stLENS1_750[408].fHigh := 66.975482; 
    stLENS1_750[409].fEnergy := 13506.855639; stLENS1_750[409].fLow := 18.700903; stLENS1_750[409].fHigh := 66.617297; 
    stLENS1_750[410].fEnergy := 13533.896382; stLENS1_750[410].fLow := 18.633075; stLENS1_750[410].fHigh := 66.261027; 
    stLENS1_750[411].fEnergy := 13560.991261; stLENS1_750[411].fLow := 18.565490; stLENS1_750[411].fHigh := 65.906663; 
    stLENS1_750[412].fEnergy := 13588.140383; stLENS1_750[412].fLow := 18.498147; stLENS1_750[412].fHigh := 65.554194; 
    stLENS1_750[413].fEnergy := 13615.343858; stLENS1_750[413].fLow := 18.431045; stLENS1_750[413].fHigh := 65.203611; 
    stLENS1_750[414].fEnergy := 13642.601795; stLENS1_750[414].fLow := 18.364183; stLENS1_750[414].fHigh := 64.854902; 
    stLENS1_750[415].fEnergy := 13669.914302; stLENS1_750[415].fLow := 18.297560; stLENS1_750[415].fHigh := 64.508057; 
    stLENS1_750[416].fEnergy := 13697.281489; stLENS1_750[416].fLow := 18.231176; stLENS1_750[416].fHigh := 64.163068; 
    stLENS1_750[417].fEnergy := 13724.703465; stLENS1_750[417].fLow := 18.165030; stLENS1_750[417].fHigh := 63.819924; 
    stLENS1_750[418].fEnergy := 13752.180339; stLENS1_750[418].fLow := 18.099120; stLENS1_750[418].fHigh := 63.478615; 
    stLENS1_750[419].fEnergy := 13779.712223; stLENS1_750[419].fLow := 18.033447; stLENS1_750[419].fHigh := 63.139131; 
    stLENS1_750[420].fEnergy := 13807.299225; stLENS1_750[420].fLow := 17.968009; stLENS1_750[420].fHigh := 62.801463; 
    stLENS1_750[421].fEnergy := 13834.941456; stLENS1_750[421].fLow := 17.902805; stLENS1_750[421].fHigh := 62.465601; 
    stLENS1_750[422].fEnergy := 13862.639028; stLENS1_750[422].fLow := 17.837834; stLENS1_750[422].fHigh := 62.131535; 
    stLENS1_750[423].fEnergy := 13890.392049; stLENS1_750[423].fLow := 17.773096; stLENS1_750[423].fHigh := 61.799255; 
    stLENS1_750[424].fEnergy := 13918.200633; stLENS1_750[424].fLow := 17.708591; stLENS1_750[424].fHigh := 61.468753; 
    stLENS1_750[425].fEnergy := 13946.064889; stLENS1_750[425].fLow := 17.644316; stLENS1_750[425].fHigh := 61.140018; 
    stLENS1_750[426].fEnergy := 13973.984929; stLENS1_750[426].fLow := 17.580271; stLENS1_750[426].fHigh := 60.813041; 
    stLENS1_750[427].fEnergy := 14001.960866; stLENS1_750[427].fLow := 17.516456; stLENS1_750[427].fHigh := 60.487813; 
    stLENS1_750[428].fEnergy := 14029.992810; stLENS1_750[428].fLow := 17.452869; stLENS1_750[428].fHigh := 60.164324; 
    stLENS1_750[429].fEnergy := 14058.080875; stLENS1_750[429].fLow := 17.389511; stLENS1_750[429].fHigh := 59.842565; 
    stLENS1_750[430].fEnergy := 14086.225171; stLENS1_750[430].fLow := 17.326379; stLENS1_750[430].fHigh := 59.522527; 
    stLENS1_750[431].fEnergy := 14114.425813; stLENS1_750[431].fLow := 17.263473; stLENS1_750[431].fHigh := 59.204200; 
    stLENS1_750[432].fEnergy := 14142.682912; stLENS1_750[432].fLow := 17.200793; stLENS1_750[432].fHigh := 58.887576; 
    stLENS1_750[433].fEnergy := 14170.996582; stLENS1_750[433].fLow := 17.138337; stLENS1_750[433].fHigh := 58.572645; 
    stLENS1_750[434].fEnergy := 14199.366936; stLENS1_750[434].fLow := 17.076105; stLENS1_750[434].fHigh := 58.259399; 
    stLENS1_750[435].fEnergy := 14227.794088; stLENS1_750[435].fLow := 17.014097; stLENS1_750[435].fHigh := 57.947827; 
    stLENS1_750[436].fEnergy := 14256.278151; stLENS1_750[436].fLow := 16.952310; stLENS1_750[436].fHigh := 57.637922; 
    stLENS1_750[437].fEnergy := 14284.819238; stLENS1_750[437].fLow := 16.890745; stLENS1_750[437].fHigh := 57.329675; 
    stLENS1_750[438].fEnergy := 14313.417466; stLENS1_750[438].fLow := 16.829400; stLENS1_750[438].fHigh := 57.023075; 
    stLENS1_750[439].fEnergy := 14342.072946; stLENS1_750[439].fLow := 16.768276; stLENS1_750[439].fHigh := 56.718116; 
    stLENS1_750[440].fEnergy := 14370.785796; stLENS1_750[440].fLow := 16.707370; stLENS1_750[440].fHigh := 56.414787; 
    stLENS1_750[441].fEnergy := 14399.556128; stLENS1_750[441].fLow := 16.646683; stLENS1_750[441].fHigh := 56.074702; 
    stLENS1_750[442].fEnergy := 14428.384059; stLENS1_750[442].fLow := 16.586213; stLENS1_750[442].fHigh := 55.801485; 
    stLENS1_750[443].fEnergy := 14457.269703; stLENS1_750[443].fLow := 16.525960; stLENS1_750[443].fHigh := 55.529694; 
    stLENS1_750[444].fEnergy := 14486.213176; stLENS1_750[444].fLow := 16.465924; stLENS1_750[444].fHigh := 55.259322; 
    stLENS1_750[445].fEnergy := 14515.214594; stLENS1_750[445].fLow := 16.406102; stLENS1_750[445].fHigh := 54.990362; 
    stLENS1_750[446].fEnergy := 14544.274073; stLENS1_750[446].fLow := 16.346495; stLENS1_750[446].fHigh := 54.722804; 
    stLENS1_750[447].fEnergy := 14573.391729; stLENS1_750[447].fLow := 16.287102; stLENS1_750[447].fHigh := 54.456643; 
    stLENS1_750[448].fEnergy := 14602.567679; stLENS1_750[448].fLow := 16.227921; stLENS1_750[448].fHigh := 54.191869; 
    stLENS1_750[449].fEnergy := 14631.802039; stLENS1_750[449].fLow := 16.168953; stLENS1_750[449].fHigh := 53.928475; 
    stLENS1_750[450].fEnergy := 14661.094926; stLENS1_750[450].fLow := 16.110196; stLENS1_750[450].fHigh := 53.666454; 
    stLENS1_750[451].fEnergy := 14690.446458; stLENS1_750[451].fLow := 16.051650; stLENS1_750[451].fHigh := 53.405798; 
    stLENS1_750[452].fEnergy := 14719.856751; stLENS1_750[452].fLow := 15.993314; stLENS1_750[452].fHigh := 53.146500; 
    stLENS1_750[453].fEnergy := 14749.325924; stLENS1_750[453].fLow := 15.935187; stLENS1_750[453].fHigh := 52.888551; 
    stLENS1_750[454].fEnergy := 14778.854094; stLENS1_750[454].fLow := 15.877269; stLENS1_750[454].fHigh := 52.631945; 
    stLENS1_750[455].fEnergy := 14808.441380; stLENS1_750[455].fLow := 15.819558; stLENS1_750[455].fHigh := 52.376675; 
    stLENS1_750[456].fEnergy := 14838.087899; stLENS1_750[456].fLow := 15.762055; stLENS1_750[456].fHigh := 52.122732; 
    stLENS1_750[457].fEnergy := 14867.793771; stLENS1_750[457].fLow := 15.704758; stLENS1_750[457].fHigh := 51.870109; 
    stLENS1_750[458].fEnergy := 14897.559114; stLENS1_750[458].fLow := 15.647666; stLENS1_750[458].fHigh := 51.618800; 
    stLENS1_750[459].fEnergy := 14927.384047; stLENS1_750[459].fLow := 15.590779; stLENS1_750[459].fHigh := 51.368797; 
    stLENS1_750[460].fEnergy := 14957.268690; stLENS1_750[460].fLow := 15.534096; stLENS1_750[460].fHigh := 51.120093; 
    stLENS1_750[461].fEnergy := 14987.213162; stLENS1_750[461].fLow := 15.477617; stLENS1_750[461].fHigh := 50.872681; 
    stLENS1_750[462].fEnergy := 15017.217582; stLENS1_750[462].fLow := 15.421340; stLENS1_750[462].fHigh := 50.626553; 
    stLENS1_750[463].fEnergy := 15047.282072; stLENS1_750[463].fLow := 15.365266; stLENS1_750[463].fHigh := 50.381703; 
    stLENS1_750[464].fEnergy := 15077.406751; stLENS1_750[464].fLow := 15.309392; stLENS1_750[464].fHigh := 50.138123; 
    stLENS1_750[465].fEnergy := 15107.591739; stLENS1_750[465].fLow := 15.253719; stLENS1_750[465].fHigh := 49.895807; 
    stLENS1_750[466].fEnergy := 15137.837158; stLENS1_750[466].fLow := 15.198246; stLENS1_750[466].fHigh := 49.654747; 
    stLENS1_750[467].fEnergy := 15168.143128; stLENS1_750[467].fLow := 15.142972; stLENS1_750[467].fHigh := 49.414937; 
    stLENS1_750[468].fEnergy := 15198.509771; stLENS1_750[468].fLow := 15.087896; stLENS1_750[468].fHigh := 49.176370; 
    stLENS1_750[469].fEnergy := 15228.937208; stLENS1_750[469].fLow := 15.033018; stLENS1_750[469].fHigh := 48.939039; 
    stLENS1_750[470].fEnergy := 15259.425560; stLENS1_750[470].fLow := 14.978337; stLENS1_750[470].fHigh := 48.702938; 
    stLENS1_750[471].fEnergy := 15289.974951; stLENS1_750[471].fLow := 14.923853; stLENS1_750[471].fHigh := 48.468058; 
    stLENS1_750[472].fEnergy := 15320.585501; stLENS1_750[472].fLow := 14.869563; stLENS1_750[472].fHigh := 48.234395; 
    stLENS1_750[473].fEnergy := 15351.257334; stLENS1_750[473].fLow := 14.815469; stLENS1_750[473].fHigh := 48.001941; 
    stLENS1_750[474].fEnergy := 15381.990571; stLENS1_750[474].fLow := 14.761569; stLENS1_750[474].fHigh := 47.770689; 
    stLENS1_750[475].fEnergy := 15412.785337; stLENS1_750[475].fLow := 14.707863; stLENS1_750[475].fHigh := 47.540633; 
    stLENS1_750[476].fEnergy := 15443.641754; stLENS1_750[476].fLow := 14.654349; stLENS1_750[476].fHigh := 47.311767; 
    stLENS1_750[477].fEnergy := 15474.559945; stLENS1_750[477].fLow := 14.601028; stLENS1_750[477].fHigh := 47.084083; 
    stLENS1_750[478].fEnergy := 15505.540035; stLENS1_750[478].fLow := 14.547898; stLENS1_750[478].fHigh := 46.857576; 
    stLENS1_750[479].fEnergy := 15536.582147; stLENS1_750[479].fLow := 14.494959; stLENS1_750[479].fHigh := 46.632238; 
    stLENS1_750[480].fEnergy := 15567.686405; stLENS1_750[480].fLow := 14.442210; stLENS1_750[480].fHigh := 46.408065; 
    stLENS1_750[481].fEnergy := 15598.852934; stLENS1_750[481].fLow := 14.389650; stLENS1_750[481].fHigh := 46.185048; 
    stLENS1_750[482].fEnergy := 15630.081858; stLENS1_750[482].fLow := 14.337280; stLENS1_750[482].fHigh := 45.963183; 
    stLENS1_750[483].fEnergy := 15661.373303; stLENS1_750[483].fLow := 14.285097; stLENS1_750[483].fHigh := 45.742462; 
    stLENS1_750[484].fEnergy := 15692.727393; stLENS1_750[484].fLow := 14.233102; stLENS1_750[484].fHigh := 45.522879; 
    stLENS1_750[485].fEnergy := 15724.144254; stLENS1_750[485].fLow := 14.181293; stLENS1_750[485].fHigh := 45.304428; 
    stLENS1_750[486].fEnergy := 15755.624012; stLENS1_750[486].fLow := 14.129671; stLENS1_750[486].fHigh := 45.087103; 
    stLENS1_750[487].fEnergy := 15787.166792; stLENS1_750[487].fLow := 14.078234; stLENS1_750[487].fHigh := 44.870899; 
    stLENS1_750[488].fEnergy := 15818.772721; stLENS1_750[488].fLow := 14.026982; stLENS1_750[488].fHigh := 44.655807; 
    stLENS1_750[489].fEnergy := 15850.441925; stLENS1_750[489].fLow := 13.975914; stLENS1_750[489].fHigh := 44.441823; 
    stLENS1_750[490].fEnergy := 15882.174531; stLENS1_750[490].fLow := 13.925030; stLENS1_750[490].fHigh := 44.228941; 
    stLENS1_750[491].fEnergy := 15913.970666; stLENS1_750[491].fLow := 13.874328; stLENS1_750[491].fHigh := 44.017155; 
    stLENS1_750[492].fEnergy := 15945.830456; stLENS1_750[492].fLow := 13.823809; stLENS1_750[492].fHigh := 43.806458; 
    stLENS1_750[493].fEnergy := 15977.754030; stLENS1_750[493].fLow := 13.773471; stLENS1_750[493].fHigh := 43.596844; 
    stLENS1_750[494].fEnergy := 16009.741515; stLENS1_750[494].fLow := 13.723314; stLENS1_750[494].fHigh := 43.388308; 
    stLENS1_750[495].fEnergy := 16041.793039; stLENS1_750[495].fLow := 13.673338; stLENS1_750[495].fHigh := 43.180844; 
    stLENS1_750[496].fEnergy := 16073.908730; stLENS1_750[496].fLow := 13.623541; stLENS1_750[496].fHigh := 42.974446; 
    stLENS1_750[497].fEnergy := 16106.088717; stLENS1_750[497].fLow := 13.573923; stLENS1_750[497].fHigh := 42.769109; 
    stLENS1_750[498].fEnergy := 16138.333128; stLENS1_750[498].fLow := 13.524483; stLENS1_750[498].fHigh := 42.564825; 
    stLENS1_750[499].fEnergy := 16170.642092; stLENS1_750[499].fLow := 13.475221; stLENS1_750[499].fHigh := 42.361591; 
    stLENS1_750[500].fEnergy := 16203.015739; stLENS1_750[500].fLow := 13.426136; stLENS1_750[500].fHigh := 42.159399; 
    stLENS1_750[501].fEnergy := 16235.454198; stLENS1_750[501].fLow := 13.377228; stLENS1_750[501].fHigh := 41.958245; 
    stLENS1_750[502].fEnergy := 16267.957599; stLENS1_750[502].fLow := 13.328496; stLENS1_750[502].fHigh := 41.758122; 
    stLENS1_750[503].fEnergy := 16300.526072; stLENS1_750[503].fLow := 13.279938; stLENS1_750[503].fHigh := 41.559025; 
    stLENS1_750[504].fEnergy := 16333.159747; stLENS1_750[504].fLow := 13.231556; stLENS1_750[504].fHigh := 41.360949; 
    stLENS1_750[505].fEnergy := 16365.858755; stLENS1_750[505].fLow := 13.183347; stLENS1_750[505].fHigh := 41.163888; 
    stLENS1_750[506].fEnergy := 16398.623226; stLENS1_750[506].fLow := 13.135312; stLENS1_750[506].fHigh := 40.967836; 
    stLENS1_750[507].fEnergy := 16431.453291; stLENS1_750[507].fLow := 13.087449; stLENS1_750[507].fHigh := 40.772789; 
    stLENS1_750[508].fEnergy := 16464.349083; stLENS1_750[508].fLow := 13.039758; stLENS1_750[508].fHigh := 40.578739; 
    stLENS1_750[509].fEnergy := 16497.310732; stLENS1_750[509].fLow := 12.992240; stLENS1_750[509].fHigh := 40.385683; 
    stLENS1_750[510].fEnergy := 16530.338370; stLENS1_750[510].fLow := 12.944891; stLENS1_750[510].fHigh := 40.193614; 
    stLENS1_750[511].fEnergy := 16563.432129; stLENS1_750[511].fLow := 12.897714; stLENS1_750[511].fHigh := 40.002528; 
    stLENS1_750[512].fEnergy := 16596.592142; stLENS1_750[512].fLow := 12.850706; stLENS1_750[512].fHigh := 39.812419; 
    stLENS1_750[513].fEnergy := 16629.818542; stLENS1_750[513].fLow := 12.803867; stLENS1_750[513].fHigh := 39.623282; 
    stLENS1_750[514].fEnergy := 16663.111461; stLENS1_750[514].fLow := 12.757196; stLENS1_750[514].fHigh := 39.435111; 
    stLENS1_750[515].fEnergy := 16696.471032; stLENS1_750[515].fLow := 12.710694; stLENS1_750[515].fHigh := 39.247901; 
    stLENS1_750[516].fEnergy := 16729.897390; stLENS1_750[516].fLow := 12.664359; stLENS1_750[516].fHigh := 39.061647; 
    stLENS1_750[517].fEnergy := 16763.390666; stLENS1_750[517].fLow := 12.618190; stLENS1_750[517].fHigh := 38.876344; 
    stLENS1_750[518].fEnergy := 16796.950997; stLENS1_750[518].fLow := 12.572188; stLENS1_750[518].fHigh := 38.691986; 
    stLENS1_750[519].fEnergy := 16830.578515; stLENS1_750[519].fLow := 12.526351; stLENS1_750[519].fHigh := 38.508570; 
    stLENS1_750[520].fEnergy := 16864.273356; stLENS1_750[520].fLow := 12.480679; stLENS1_750[520].fHigh := 38.326088; 
    stLENS1_750[521].fEnergy := 16898.035654; stLENS1_750[521].fLow := 12.435171; stLENS1_750[521].fHigh := 38.144537; 
    stLENS1_750[522].fEnergy := 16931.865544; stLENS1_750[522].fLow := 12.389828; stLENS1_750[522].fHigh := 37.963912; 
    stLENS1_750[523].fEnergy := 16965.763161; stLENS1_750[523].fLow := 12.344647; stLENS1_750[523].fHigh := 37.784207; 
    stLENS1_750[524].fEnergy := 16999.728641; stLENS1_750[524].fLow := 12.299629; stLENS1_750[524].fHigh := 37.605417; 
    stLENS1_750[525].fEnergy := 17033.762121; stLENS1_750[525].fLow := 12.254773; stLENS1_750[525].fHigh := 37.427538; 
    stLENS1_750[526].fEnergy := 17067.863735; stLENS1_750[526].fLow := 12.210079; stLENS1_750[526].fHigh := 37.250564; 
    stLENS1_750[527].fEnergy := 17102.033621; stLENS1_750[527].fLow := 12.165545; stLENS1_750[527].fHigh := 37.074491; 
    stLENS1_750[528].fEnergy := 17136.271915; stLENS1_750[528].fLow := 12.121172; stLENS1_750[528].fHigh := 36.899314; 
    stLENS1_750[529].fEnergy := 17170.578755; stLENS1_750[529].fLow := 12.076958; stLENS1_750[529].fHigh := 36.725027; 
    stLENS1_750[530].fEnergy := 17204.954276; stLENS1_750[530].fLow := 12.032904; stLENS1_750[530].fHigh := 36.551627; 
    stLENS1_750[531].fEnergy := 17239.398618; stLENS1_750[531].fLow := 11.989008; stLENS1_750[531].fHigh := 36.379108; 
    stLENS1_750[532].fEnergy := 17273.911917; stLENS1_750[532].fLow := 11.945270; stLENS1_750[532].fHigh := 36.207466; 
    stLENS1_750[533].fEnergy := 17308.494311; stLENS1_750[533].fLow := 11.901690; stLENS1_750[533].fHigh := 36.036696; 
    stLENS1_750[534].fEnergy := 17343.145940; stLENS1_750[534].fLow := 11.858267; stLENS1_750[534].fHigh := 35.866792; 
    stLENS1_750[535].fEnergy := 17377.866941; stLENS1_750[535].fLow := 11.815000; stLENS1_750[535].fHigh := 35.697752; 
    stLENS1_750[536].fEnergy := 17412.657454; stLENS1_750[536].fLow := 11.771889; stLENS1_750[536].fHigh := 35.529569; 
    stLENS1_750[537].fEnergy := 17447.517618; stLENS1_750[537].fLow := 11.728933; stLENS1_750[537].fHigh := 35.362239; 
    stLENS1_750[538].fEnergy := 17482.447571; stLENS1_750[538].fLow := 11.686132; stLENS1_750[538].fHigh := 35.195759; 
    stLENS1_750[539].fEnergy := 17517.447455; stLENS1_750[539].fLow := 11.643485; stLENS1_750[539].fHigh := 35.030122; 
    stLENS1_750[540].fEnergy := 17552.517408; stLENS1_750[540].fLow := 11.600992; stLENS1_750[540].fHigh := 34.865325; 
    stLENS1_750[541].fEnergy := 17587.657571; stLENS1_750[541].fLow := 11.558652; stLENS1_750[541].fHigh := 34.701362; 
    stLENS1_750[542].fEnergy := 17622.868085; stLENS1_750[542].fLow := 11.516464; stLENS1_750[542].fHigh := 34.538231; 
    stLENS1_750[543].fEnergy := 17658.149090; stLENS1_750[543].fLow := 11.474428; stLENS1_750[543].fHigh := 34.375925; 
    stLENS1_750[544].fEnergy := 17693.500728; stLENS1_750[544].fLow := 11.432544; stLENS1_750[544].fHigh := 34.214441; 
    stLENS1_750[545].fEnergy := 17728.923140; stLENS1_750[545].fLow := 11.390810; stLENS1_750[545].fHigh := 34.053775; 
    stLENS1_750[546].fEnergy := 17764.416468; stLENS1_750[546].fLow := 11.349227; stLENS1_750[546].fHigh := 33.893921; 
    stLENS1_750[547].fEnergy := 17799.980854; stLENS1_750[547].fLow := 11.307794; stLENS1_750[547].fHigh := 33.734875; 
    stLENS1_750[548].fEnergy := 17835.616439; stLENS1_750[548].fLow := 11.266510; stLENS1_750[548].fHigh := 33.576634; 
    stLENS1_750[549].fEnergy := 17871.323367; stLENS1_750[549].fLow := 11.225375; stLENS1_750[549].fHigh := 33.419192; 
    stLENS1_750[550].fEnergy := 17907.101780; stLENS1_750[550].fLow := 11.184388; stLENS1_750[550].fHigh := 33.262547; 
    stLENS1_750[551].fEnergy := 17942.951822; stLENS1_750[551].fLow := 11.143549; stLENS1_750[551].fHigh := 33.106692; 
    stLENS1_750[552].fEnergy := 17978.873635; stLENS1_750[552].fLow := 11.102857; stLENS1_750[552].fHigh := 32.951624; 
    stLENS1_750[553].fEnergy := 18014.867364; stLENS1_750[553].fLow := 11.062312; stLENS1_750[553].fHigh := 32.797339; 
    stLENS1_750[554].fEnergy := 18050.933153; stLENS1_750[554].fLow := 11.021912; stLENS1_750[554].fHigh := 32.643833; 
    stLENS1_750[555].fEnergy := 18087.071145; stLENS1_750[555].fLow := 10.981659; stLENS1_750[555].fHigh := 32.491101; 
    stLENS1_750[556].fEnergy := 18123.281486; stLENS1_750[556].fLow := 10.941550; stLENS1_750[556].fHigh := 32.339140; 
    stLENS1_750[557].fEnergy := 18159.564319; stLENS1_750[557].fLow := 10.901587; stLENS1_750[557].fHigh := 32.187944; 
    stLENS1_750[558].fEnergy := 18195.919791; stLENS1_750[558].fLow := 10.861767; stLENS1_750[558].fHigh := 32.037511; 
    stLENS1_750[559].fEnergy := 18232.348047; stLENS1_750[559].fLow := 10.822091; stLENS1_750[559].fHigh := 31.887835; 
    stLENS1_750[560].fEnergy := 18268.849232; stLENS1_750[560].fLow := 10.782557; stLENS1_750[560].fHigh := 31.738914; 
    stLENS1_750[561].fEnergy := 18305.423493; stLENS1_750[561].fLow := 10.743167; stLENS1_750[561].fHigh := 31.590742; 
    stLENS1_750[562].fEnergy := 18342.070975; stLENS1_750[562].fLow := 10.703918; stLENS1_750[562].fHigh := 31.443317; 
    stLENS1_750[563].fEnergy := 18378.791826; stLENS1_750[563].fLow := 10.664811; stLENS1_750[563].fHigh := 31.296633; 
    stLENS1_750[564].fEnergy := 18415.586191; stLENS1_750[564].fLow := 10.625845; stLENS1_750[564].fHigh := 31.150687; 
    stLENS1_750[565].fEnergy := 18452.454219; stLENS1_750[565].fLow := 10.587020; stLENS1_750[565].fHigh := 31.005475; 
    stLENS1_750[566].fEnergy := 18489.396057; stLENS1_750[566].fLow := 10.548334; stLENS1_750[566].fHigh := 30.860993; 
    stLENS1_750[567].fEnergy := 18526.411853; stLENS1_750[567].fLow := 10.509788; stLENS1_750[567].fHigh := 30.717237; 
    stLENS1_750[568].fEnergy := 18563.501754; stLENS1_750[568].fLow := 10.471381; stLENS1_750[568].fHigh := 30.574204; 
    stLENS1_750[569].fEnergy := 18600.665909; stLENS1_750[569].fLow := 10.433113; stLENS1_750[569].fHigh := 30.431889; 
    stLENS1_750[570].fEnergy := 18637.904467; stLENS1_750[570].fLow := 10.394983; stLENS1_750[570].fHigh := 30.290288; 
    stLENS1_750[571].fEnergy := 18675.217577; stLENS1_750[571].fLow := 10.356990; stLENS1_750[571].fHigh := 30.149399; 
    stLENS1_750[572].fEnergy := 18712.605388; stLENS1_750[572].fLow := 10.319134; stLENS1_750[572].fHigh := 30.009216; 
    stLENS1_750[573].fEnergy := 18750.068048; stLENS1_750[573].fLow := 10.281415; stLENS1_750[573].fHigh := 29.869737; 
    stLENS1_750[574].fEnergy := 18787.605710; stLENS1_750[574].fLow := 10.243832; stLENS1_750[574].fHigh := 29.730957; 
    stLENS1_750[575].fEnergy := 18825.218521; stLENS1_750[575].fLow := 10.206385; stLENS1_750[575].fHigh := 29.592873; 
    stLENS1_750[576].fEnergy := 18862.906634; stLENS1_750[576].fLow := 10.169072; stLENS1_750[576].fHigh := 29.455481; 
    stLENS1_750[577].fEnergy := 18900.670198; stLENS1_750[577].fLow := 10.131895; stLENS1_750[577].fHigh := 29.318777; 
    stLENS1_750[578].fEnergy := 18938.509365; stLENS1_750[578].fLow := 10.094851; stLENS1_750[578].fHigh := 29.182758; 
    stLENS1_750[579].fEnergy := 18976.424286; stLENS1_750[579].fLow := 10.057941; stLENS1_750[579].fHigh := 29.047420; 
    stLENS1_750[580].fEnergy := 19014.415113; stLENS1_750[580].fLow := 10.021165; stLENS1_750[580].fHigh := 28.912759; 
    stLENS1_750[581].fEnergy := 19052.481997; stLENS1_750[581].fLow := 9.984521; stLENS1_750[581].fHigh := 28.778773; 
    stLENS1_750[582].fEnergy := 19090.625092; stLENS1_750[582].fLow := 9.948009; stLENS1_750[582].fHigh := 28.645456; 
    stLENS1_750[583].fEnergy := 19128.844549; stLENS1_750[583].fLow := 9.911629; stLENS1_750[583].fHigh := 28.512806; 
    stLENS1_750[584].fEnergy := 19167.140521; stLENS1_750[584].fLow := 9.875381; stLENS1_750[584].fHigh := 28.380820; 
    stLENS1_750[585].fEnergy := 19205.513162; stLENS1_750[585].fLow := 9.839263; stLENS1_750[585].fHigh := 28.249492; 
    stLENS1_750[586].fEnergy := 19243.962625; stLENS1_750[586].fLow := 9.803276; stLENS1_750[586].fHigh := 28.118821; 
    stLENS1_750[587].fEnergy := 19282.489064; stLENS1_750[587].fLow := 9.767418; stLENS1_750[587].fHigh := 27.988803; 
    stLENS1_750[588].fEnergy := 19321.092632; stLENS1_750[588].fLow := 9.731690; stLENS1_750[588].fHigh := 27.859434; 
    stLENS1_750[589].fEnergy := 19359.773486; stLENS1_750[589].fLow := 9.696092; stLENS1_750[589].fHigh := 27.730711; 
    stLENS1_750[590].fEnergy := 19398.531778; stLENS1_750[590].fLow := 9.660621; stLENS1_750[590].fHigh := 27.602629; 
    stLENS1_750[591].fEnergy := 19437.367665; stLENS1_750[591].fLow := 9.625279; stLENS1_750[591].fHigh := 27.475187; 
    stLENS1_750[592].fEnergy := 19476.281301; stLENS1_750[592].fLow := 9.590064; stLENS1_750[592].fHigh := 27.348380; 
    stLENS1_750[593].fEnergy := 19515.272842; stLENS1_750[593].fLow := 9.554977; stLENS1_750[593].fHigh := 27.222206; 
    stLENS1_750[594].fEnergy := 19554.342444; stLENS1_750[594].fLow := 9.520016; stLENS1_750[594].fHigh := 27.096660; 
    stLENS1_750[595].fEnergy := 19593.490264; stLENS1_750[595].fLow := 9.485182; stLENS1_750[595].fHigh := 26.971739; 
    stLENS1_750[596].fEnergy := 19632.716457; stLENS1_750[596].fLow := 9.450473; stLENS1_750[596].fHigh := 26.847441; 
    stLENS1_750[597].fEnergy := 19672.021182; stLENS1_750[597].fLow := 9.415890; stLENS1_750[597].fHigh := 26.723762; 
    stLENS1_750[598].fEnergy := 19711.404594; stLENS1_750[598].fLow := 9.381431; stLENS1_750[598].fHigh := 26.600698; 
    stLENS1_750[599].fEnergy := 19750.866853; stLENS1_750[599].fLow := 9.347097; stLENS1_750[599].fHigh := 26.478246; 
    stLENS1_750[600].fEnergy := 19790.408115; stLENS1_750[600].fLow := 9.312888; stLENS1_750[600].fHigh := 26.356404; 
    stLENS1_750[601].fEnergy := 19830.028538; stLENS1_750[601].fLow := 9.278801; stLENS1_750[601].fHigh := 26.235167; 
    stLENS1_750[602].fEnergy := 19869.728282; stLENS1_750[602].fLow := 9.244838; stLENS1_750[602].fHigh := 26.114533; 
    stLENS1_750[603].fEnergy := 19909.507504; stLENS1_750[603].fLow := 9.210998; stLENS1_750[603].fHigh := 25.994498; 
    stLENS1_750[604].fEnergy := 19949.366365; stLENS1_750[604].fLow := 9.177280; stLENS1_750[604].fHigh := 25.875060; 
    stLENS1_750[605].fEnergy := 19989.305023; stLENS1_750[605].fLow := 9.143683; stLENS1_750[605].fHigh := 25.756215; 
    stLENS1_750[606].fEnergy := 20029.323638; stLENS1_750[606].fLow := 9.110208; stLENS1_750[606].fHigh := 25.637960; 
    stLENS1_750[607].fEnergy := 20069.422371; stLENS1_750[607].fLow := 9.076854; stLENS1_750[607].fHigh := 25.520292; 
    stLENS1_750[608].fEnergy := 20109.601381; stLENS1_750[608].fLow := 9.043621; stLENS1_750[608].fHigh := 25.403207; 
    stLENS1_750[609].fEnergy := 20149.860830; stLENS1_750[609].fLow := 9.010508; stLENS1_750[609].fHigh := 25.286704; 
    stLENS1_750[610].fEnergy := 20190.200878; stLENS1_750[610].fLow := 8.977514; stLENS1_750[610].fHigh := 25.170778; 
    stLENS1_750[611].fEnergy := 20230.621687; stLENS1_750[611].fLow := 8.944640; stLENS1_750[611].fHigh := 25.055426; 
    stLENS1_750[612].fEnergy := 20271.123419; stLENS1_750[612].fLow := 8.911884; stLENS1_750[612].fHigh := 24.940646; 
    stLENS1_750[613].fEnergy := 20311.706235; stLENS1_750[613].fLow := 8.879247; stLENS1_750[613].fHigh := 24.826435; 
    stLENS1_750[614].fEnergy := 20352.370298; stLENS1_750[614].fLow := 8.846728; stLENS1_750[614].fHigh := 24.712789; 
    stLENS1_750[615].fEnergy := 20393.115770; stLENS1_750[615].fLow := 8.814326; stLENS1_750[615].fHigh := 24.599706; 
    stLENS1_750[616].fEnergy := 20433.942815; stLENS1_750[616].fLow := 8.782042; stLENS1_750[616].fHigh := 24.487182; 
    stLENS1_750[617].fEnergy := 20474.851596; stLENS1_750[617].fLow := 8.749874; stLENS1_750[617].fHigh := 24.375215; 
    stLENS1_750[618].fEnergy := 20515.842276; stLENS1_750[618].fLow := 8.717823; stLENS1_750[618].fHigh := 24.263802; 
    stLENS1_750[619].fEnergy := 20556.915020; stLENS1_750[619].fLow := 8.685887; stLENS1_750[619].fHigh := 24.152940; 
    stLENS1_750[620].fEnergy := 20598.069991; stLENS1_750[620].fLow := 8.654067; stLENS1_750[620].fHigh := 24.042626; 
    stLENS1_750[621].fEnergy := 20639.307355; stLENS1_750[621].fLow := 8.622362; stLENS1_750[621].fHigh := 23.932856; 
    stLENS1_750[622].fEnergy := 20680.627276; stLENS1_750[622].fLow := 8.590772; stLENS1_750[622].fHigh := 23.823629; 
    stLENS1_750[623].fEnergy := 20722.029919; stLENS1_750[623].fLow := 8.559296; stLENS1_750[623].fHigh := 23.714941; 
    stLENS1_750[624].fEnergy := 20763.515451; stLENS1_750[624].fLow := 8.527934; stLENS1_750[624].fHigh := 23.606790; 
    stLENS1_750[625].fEnergy := 20805.084036; stLENS1_750[625].fLow := 8.496685; stLENS1_750[625].fHigh := 23.499172; 
    stLENS1_750[626].fEnergy := 20846.735842; stLENS1_750[626].fLow := 8.465549; stLENS1_750[626].fHigh := 23.392086; 
    stLENS1_750[627].fEnergy := 20888.471035; stLENS1_750[627].fLow := 8.434526; stLENS1_750[627].fHigh := 23.285527; 
    stLENS1_750[628].fEnergy := 20930.289782; stLENS1_750[628].fLow := 8.403615; stLENS1_750[628].fHigh := 23.179494; 
    stLENS1_750[629].fEnergy := 20972.192250; stLENS1_750[629].fLow := 8.372816; stLENS1_750[629].fHigh := 23.073983; 
    stLENS1_750[630].fEnergy := 21014.178607; stLENS1_750[630].fLow := 8.342129; stLENS1_750[630].fHigh := 22.968992; 
    stLENS1_750[631].fEnergy := 21056.249021; stLENS1_750[631].fLow := 8.311552; stLENS1_750[631].fHigh := 22.864518; 
    stLENS1_750[632].fEnergy := 21098.403659; stLENS1_750[632].fLow := 8.281086; stLENS1_750[632].fHigh := 22.760559; 
    stLENS1_750[633].fEnergy := 21140.642692; stLENS1_750[633].fLow := 8.250730; stLENS1_750[633].fHigh := 22.657111; 
    stLENS1_750[634].fEnergy := 21182.966286; stLENS1_750[634].fLow := 8.220485; stLENS1_750[634].fHigh := 22.554172; 
    stLENS1_750[635].fEnergy := 21225.374613; stLENS1_750[635].fLow := 8.190348; stLENS1_750[635].fHigh := 22.451740; 
    stLENS1_750[636].fEnergy := 21267.867841; stLENS1_750[636].fLow := 8.160321; stLENS1_750[636].fHigh := 22.349811; 
    stLENS1_750[637].fEnergy := 21310.446141; stLENS1_750[637].fLow := 8.130402; stLENS1_750[637].fHigh := 22.248384; 
    stLENS1_750[638].fEnergy := 21353.109683; stLENS1_750[638].fLow := 8.100592; stLENS1_750[638].fHigh := 22.147455; 
    stLENS1_750[639].fEnergy := 21395.858637; stLENS1_750[639].fLow := 8.070889; stLENS1_750[639].fHigh := 22.047021; 
    stLENS1_750[640].fEnergy := 21438.693174; stLENS1_750[640].fLow := 8.041294; stLENS1_750[640].fHigh := 21.947081; 
    stLENS1_750[641].fEnergy := 21481.613467; stLENS1_750[641].fLow := 8.011806; stLENS1_750[641].fHigh := 21.847632; 
    stLENS1_750[642].fEnergy := 21524.619686; stLENS1_750[642].fLow := 7.982425; stLENS1_750[642].fHigh := 21.748670; 
    stLENS1_750[643].fEnergy := 21567.712003; stLENS1_750[643].fLow := 7.953150; stLENS1_750[643].fHigh := 21.650194; 
    stLENS1_750[644].fEnergy := 21610.890591; stLENS1_750[644].fLow := 7.923981; stLENS1_750[644].fHigh := 21.552201; 
    stLENS1_750[645].fEnergy := 21654.155623; stLENS1_750[645].fLow := 7.894918; stLENS1_750[645].fHigh := 21.454689; 
    stLENS1_750[646].fEnergy := 21697.507271; stLENS1_750[646].fLow := 7.865960; stLENS1_750[646].fHigh := 21.357655; 
    stLENS1_750[647].fEnergy := 21740.945710; stLENS1_750[647].fLow := 7.837107; stLENS1_750[647].fHigh := 21.261096; 
    stLENS1_750[648].fEnergy := 21784.471112; stLENS1_750[648].fLow := 7.808358; stLENS1_750[648].fHigh := 21.165010; 
    stLENS1_750[649].fEnergy := 21828.083652; stLENS1_750[649].fLow := 7.779714; stLENS1_750[649].fHigh := 21.069394; 
    stLENS1_750[650].fEnergy := 21871.783505; stLENS1_750[650].fLow := 7.751173; stLENS1_750[650].fHigh := 20.974247; 
    stLENS1_750[651].fEnergy := 21915.570845; stLENS1_750[651].fLow := 7.722736; stLENS1_750[651].fHigh := 20.879565; 
    stLENS1_750[652].fEnergy := 21959.445847; stLENS1_750[652].fLow := 7.694401; stLENS1_750[652].fHigh := 20.785347; 
    stLENS1_750[653].fEnergy := 22003.408687; stLENS1_750[653].fLow := 7.666169; stLENS1_750[653].fHigh := 20.691589; 
    stLENS1_750[654].fEnergy := 22047.459540; stLENS1_750[654].fLow := 7.638040; stLENS1_750[654].fHigh := 20.598290; 
    stLENS1_750[655].fEnergy := 22091.598584; stLENS1_750[655].fLow := 7.610012; stLENS1_750[655].fHigh := 20.505446; 
    stLENS1_750[656].fEnergy := 22135.825994; stLENS1_750[656].fLow := 7.582086; stLENS1_750[656].fHigh := 20.413057; 
    stLENS1_750[657].fEnergy := 22180.141947; stLENS1_750[657].fLow := 7.554261; stLENS1_750[657].fHigh := 20.321118; 
    stLENS1_750[658].fEnergy := 22224.546620; stLENS1_750[658].fLow := 7.526537; stLENS1_750[658].fHigh := 20.229629; 
    stLENS1_750[659].fEnergy := 22269.040192; stLENS1_750[659].fLow := 7.498913; stLENS1_750[659].fHigh := 20.138586; 
    stLENS1_750[660].fEnergy := 22313.622841; stLENS1_750[660].fLow := 7.471389; stLENS1_750[660].fHigh := 20.047987; 
    stLENS1_750[661].fEnergy := 22358.294743; stLENS1_750[661].fLow := 7.443965; stLENS1_750[661].fHigh := 19.957830; 
    stLENS1_750[662].fEnergy := 22403.056079; stLENS1_750[662].fLow := 7.416641; stLENS1_750[662].fHigh := 19.868113; 
    stLENS1_750[663].fEnergy := 22447.907027; stLENS1_750[663].fLow := 7.389415; stLENS1_750[663].fHigh := 19.778834; 
    stLENS1_750[664].fEnergy := 22492.847767; stLENS1_750[664].fLow := 7.362288; stLENS1_750[664].fHigh := 19.689989; 
    stLENS1_750[665].fEnergy := 22537.878478; stLENS1_750[665].fLow := 7.335260; stLENS1_750[665].fHigh := 19.601577; 
    stLENS1_750[666].fEnergy := 22582.999341; stLENS1_750[666].fLow := 7.308329; stLENS1_750[666].fHigh := 19.513596; 
    stLENS1_750[667].fEnergy := 22628.210536; stLENS1_750[667].fLow := 7.281496; stLENS1_750[667].fHigh := 19.426043; 
    stLENS1_750[668].fEnergy := 22673.512244; stLENS1_750[668].fLow := 7.254760; stLENS1_750[668].fHigh := 19.338916; 
    stLENS1_750[669].fEnergy := 22718.904645; stLENS1_750[669].fLow := 7.228121; stLENS1_750[669].fHigh := 19.252213; 
    stLENS1_750[670].fEnergy := 22764.387923; stLENS1_750[670].fLow := 7.201579; stLENS1_750[670].fHigh := 19.165932; 
    stLENS1_750[671].fEnergy := 22809.962258; stLENS1_750[671].fLow := 7.175133; stLENS1_750[671].fHigh := 19.080071; 
    stLENS1_750[672].fEnergy := 22855.627833; stLENS1_750[672].fLow := 7.148783; stLENS1_750[672].fHigh := 18.994627; 
    stLENS1_750[673].fEnergy := 22901.384830; stLENS1_750[673].fLow := 7.122528; stLENS1_750[673].fHigh := 18.909598; 
    stLENS1_750[674].fEnergy := 22947.233433; stLENS1_750[674].fLow := 7.096368; stLENS1_750[674].fHigh := 18.824982; 
    stLENS1_750[675].fEnergy := 22993.173825; stLENS1_750[675].fLow := 7.070304; stLENS1_750[675].fHigh := 18.740777; 
    stLENS1_750[676].fEnergy := 23039.206190; stLENS1_750[676].fLow := 7.044334; stLENS1_750[676].fHigh := 18.656980; 
    stLENS1_750[677].fEnergy := 23085.330711; stLENS1_750[677].fLow := 7.018458; stLENS1_750[677].fHigh := 18.573591; 
    stLENS1_750[678].fEnergy := 23131.547574; stLENS1_750[678].fLow := 6.992676; stLENS1_750[678].fHigh := 18.490606; 
    stLENS1_750[679].fEnergy := 23177.856963; stLENS1_750[679].fLow := 6.966987; stLENS1_750[679].fHigh := 18.408023; 
    stLENS1_750[680].fEnergy := 23224.259064; stLENS1_750[680].fLow := 6.941391; stLENS1_750[680].fHigh := 18.325841; 
    stLENS1_750[681].fEnergy := 23270.754061; stLENS1_750[681].fLow := 6.915889; stLENS1_750[681].fHigh := 18.244057; 
    stLENS1_750[682].fEnergy := 23317.342142; stLENS1_750[682].fLow := 6.890479; stLENS1_750[682].fHigh := 18.162669; 
    stLENS1_750[683].fEnergy := 23364.023492; stLENS1_750[683].fLow := 6.865161; stLENS1_750[683].fHigh := 18.081676; 
    stLENS1_750[684].fEnergy := 23410.798298; stLENS1_750[684].fLow := 6.839934; stLENS1_750[684].fHigh := 18.001075; 
    stLENS1_750[685].fEnergy := 23457.666748; stLENS1_750[685].fLow := 6.814800; stLENS1_750[685].fHigh := 17.920864; 
    stLENS1_750[686].fEnergy := 23504.629028; stLENS1_750[686].fLow := 6.789756; stLENS1_750[686].fHigh := 17.841041; 
    stLENS1_750[687].fEnergy := 23551.685327; stLENS1_750[687].fLow := 6.764804; stLENS1_750[687].fHigh := 17.761604; 
    stLENS1_750[688].fEnergy := 23598.835832; stLENS1_750[688].fLow := 6.739942; stLENS1_750[688].fHigh := 17.682551; 
    stLENS1_750[689].fEnergy := 23646.080733; stLENS1_750[689].fLow := 6.715170; stLENS1_750[689].fHigh := 17.603881; 
    stLENS1_750[690].fEnergy := 23693.420218; stLENS1_750[690].fLow := 6.690488; stLENS1_750[690].fHigh := 17.525590; 
    stLENS1_750[691].fEnergy := 23740.854477; stLENS1_750[691].fLow := 6.665895; stLENS1_750[691].fHigh := 17.447678; 
    stLENS1_750[692].fEnergy := 23788.383699; stLENS1_750[692].fLow := 6.641392; stLENS1_750[692].fHigh := 17.370142; 
    stLENS1_750[693].fEnergy := 23836.008075; stLENS1_750[693].fLow := 6.616978; stLENS1_750[693].fHigh := 17.292981; 
    stLENS1_750[694].fEnergy := 23883.727795; stLENS1_750[694].fLow := 6.592652; stLENS1_750[694].fHigh := 17.216192; 
    stLENS1_750[695].fEnergy := 23931.543050; stLENS1_750[695].fLow := 6.568415; stLENS1_750[695].fHigh := 17.139773; 
    stLENS1_750[696].fEnergy := 23979.454031; stLENS1_750[696].fLow := 6.544265; stLENS1_750[696].fHigh := 17.063723; 
    stLENS1_750[697].fEnergy := 24027.460930; stLENS1_750[697].fLow := 6.520203; stLENS1_750[697].fHigh := 16.988040; 
    stLENS1_750[698].fEnergy := 24075.563939; stLENS1_750[698].fLow := 6.496229; stLENS1_750[698].fHigh := 16.912721; 
    stLENS1_750[699].fEnergy := 24123.763250; stLENS1_750[699].fLow := 6.472342; stLENS1_750[699].fHigh := 16.837766; 
    stLENS1_750[700].fEnergy := 24172.059056; stLENS1_750[700].fLow := 6.448541; stLENS1_750[700].fHigh := 16.763171; 
    stLENS1_750[701].fEnergy := 24220.451551; stLENS1_750[701].fLow := 6.424827; stLENS1_750[701].fHigh := 16.688936; 
    stLENS1_750[702].fEnergy := 24268.940927; stLENS1_750[702].fLow := 6.401198; stLENS1_750[702].fHigh := 16.615058; 
    stLENS1_750[703].fEnergy := 24317.527379; stLENS1_750[703].fLow := 6.377656; stLENS1_750[703].fHigh := 16.541535; 
    stLENS1_750[704].fEnergy := 24366.211101; stLENS1_750[704].fLow := 6.354199; stLENS1_750[704].fHigh := 16.468367; 
    stLENS1_750[705].fEnergy := 24414.992288; stLENS1_750[705].fLow := 6.330827; stLENS1_750[705].fHigh := 16.395550; 
    stLENS1_750[706].fEnergy := 24463.871136; stLENS1_750[706].fLow := 6.307540; stLENS1_750[706].fHigh := 16.323083; 
    stLENS1_750[707].fEnergy := 24512.847838; stLENS1_750[707].fLow := 6.284338; stLENS1_750[707].fHigh := 16.250965; 
    stLENS1_750[708].fEnergy := 24561.922592; stLENS1_750[708].fLow := 6.261220; stLENS1_750[708].fHigh := 16.179193; 
    stLENS1_750[709].fEnergy := 24611.095594; stLENS1_750[709].fLow := 6.238186; stLENS1_750[709].fHigh := 16.107765; 
    stLENS1_750[710].fEnergy := 24660.367040; stLENS1_750[710].fLow := 6.215235; stLENS1_750[710].fHigh := 16.036681; 
    stLENS1_750[711].fEnergy := 24709.737128; stLENS1_750[711].fLow := 6.192368; stLENS1_750[711].fHigh := 15.965938; 
    stLENS1_750[712].fEnergy := 24759.206055; stLENS1_750[712].fLow := 6.169584; stLENS1_750[712].fHigh := 15.895534; 
    stLENS1_750[713].fEnergy := 24808.774018; stLENS1_750[713].fLow := 6.146883; stLENS1_750[713].fHigh := 15.825468; 
    stLENS1_750[714].fEnergy := 24858.441217; stLENS1_750[714].fLow := 6.124264; stLENS1_750[714].fHigh := 15.755738; 
    stLENS1_750[715].fEnergy := 24908.207849; stLENS1_750[715].fLow := 6.101727; stLENS1_750[715].fHigh := 15.686342; 
    stLENS1_750[716].fEnergy := 24958.074115; stLENS1_750[716].fLow := 6.079273; stLENS1_750[716].fHigh := 15.617279; 
    stLENS1_750[717].fEnergy := 25008.040212; stLENS1_750[717].fLow := 6.056899; stLENS1_750[717].fHigh := 15.548547; 
    stLENS1_750[718].fEnergy := 25058.106342; stLENS1_750[718].fLow := 6.034607; stLENS1_750[718].fHigh := 15.480143; 
    stLENS1_750[719].fEnergy := 25108.272705; stLENS1_750[719].fLow := 6.012397; stLENS1_750[719].fHigh := 15.412068; 
    stLENS1_750[720].fEnergy := 25158.539500; stLENS1_750[720].fLow := 5.990266; stLENS1_750[720].fHigh := 15.344318; 
    stLENS1_750[721].fEnergy := 25208.906930; stLENS1_750[721].fLow := 5.968217; stLENS1_750[721].fHigh := 15.276892; 
    stLENS1_750[722].fEnergy := 25259.375195; stLENS1_750[722].fLow := 5.946247; stLENS1_750[722].fHigh := 15.209788; 
    stLENS1_750[723].fEnergy := 25309.944498; stLENS1_750[723].fLow := 5.924357; stLENS1_750[723].fHigh := 15.143006; 
    stLENS1_750[724].fEnergy := 25360.615041; stLENS1_750[724].fLow := 5.902547; stLENS1_750[724].fHigh := 15.076543; 
    stLENS1_750[725].fEnergy := 25411.387026; stLENS1_750[725].fLow := 5.880816; stLENS1_750[725].fHigh := 15.010397; 
    stLENS1_750[726].fEnergy := 25462.260656; stLENS1_750[726].fLow := 5.859164; stLENS1_750[726].fHigh := 14.944567; 
    stLENS1_750[727].fEnergy := 25513.236136; stLENS1_750[727].fLow := 5.837590; stLENS1_750[727].fHigh := 14.879051; 
    stLENS1_750[728].fEnergy := 25564.313669; stLENS1_750[728].fLow := 5.816096; stLENS1_750[728].fHigh := 14.813848; 
    stLENS1_750[729].fEnergy := 25615.493459; stLENS1_750[729].fLow := 5.794679; stLENS1_750[729].fHigh := 14.748957; 
    stLENS1_750[730].fEnergy := 25666.775711; stLENS1_750[730].fLow := 5.773340; stLENS1_750[730].fHigh := 14.684375; 
    stLENS1_750[731].fEnergy := 25718.160630; stLENS1_750[731].fLow := 5.752079; stLENS1_750[731].fHigh := 14.620100; 
    stLENS1_750[732].fEnergy := 25769.648422; stLENS1_750[732].fLow := 5.730895; stLENS1_750[732].fHigh := 14.556133; 
    stLENS1_750[733].fEnergy := 25821.239293; stLENS1_750[733].fLow := 5.709788; stLENS1_750[733].fHigh := 14.492470; 
    stLENS1_750[734].fEnergy := 25872.933448; stLENS1_750[734].fLow := 5.688757; stLENS1_750[734].fHigh := 14.429110; 
    stLENS1_750[735].fEnergy := 25924.731096; stLENS1_750[735].fLow := 5.667804; stLENS1_750[735].fHigh := 14.366052; 
    stLENS1_750[736].fEnergy := 25976.632442; stLENS1_750[736].fLow := 5.646926; stLENS1_750[736].fHigh := 14.303294; 
    stLENS1_750[737].fEnergy := 26028.637695; stLENS1_750[737].fLow := 5.626124; stLENS1_750[737].fHigh := 14.240835; 
    stLENS1_750[738].fEnergy := 26080.747062; stLENS1_750[738].fLow := 5.605398; stLENS1_750[738].fHigh := 14.178673; 
    stLENS1_750[739].fEnergy := 26132.960752; stLENS1_750[739].fLow := 5.584748; stLENS1_750[739].fHigh := 14.116807; 
    stLENS1_750[740].fEnergy := 26185.278975; stLENS1_750[740].fLow := 5.564172; stLENS1_750[740].fHigh := 14.055235; 
    stLENS1_750[741].fEnergy := 26237.701938; stLENS1_750[741].fLow := 5.543671; stLENS1_750[741].fHigh := 13.993956; 
    stLENS1_750[742].fEnergy := 26290.229852; stLENS1_750[742].fLow := 5.523245; stLENS1_750[742].fHigh := 13.932967; 
    stLENS1_750[743].fEnergy := 26342.862928; stLENS1_750[743].fLow := 5.502894; stLENS1_750[743].fHigh := 13.872269; 
    stLENS1_750[744].fEnergy := 26395.601374; stLENS1_750[744].fLow := 5.482616; stLENS1_750[744].fHigh := 13.811858; 
    stLENS1_750[745].fEnergy := 26448.445404; stLENS1_750[745].fLow := 5.462412; stLENS1_750[745].fHigh := 13.751735; 
    stLENS1_750[746].fEnergy := 26501.395226; stLENS1_750[746].fLow := 5.442281; stLENS1_750[746].fHigh := 13.691896; 
    stLENS1_750[747].fEnergy := 26554.451055; stLENS1_750[747].fLow := 5.422224; stLENS1_750[747].fHigh := 13.632342; 
    stLENS1_750[748].fEnergy := 26607.613102; stLENS1_750[748].fLow := 5.402240; stLENS1_750[748].fHigh := 13.573070; 
    stLENS1_750[749].fEnergy := 26660.881578; stLENS1_750[749].fLow := 5.382328; stLENS1_750[749].fHigh := 13.514079; 
    stLENS1_750[750].fEnergy := 26714.256699; stLENS1_750[750].fLow := 5.362489; stLENS1_750[750].fHigh := 13.455367; 
    stLENS1_750[751].fEnergy := 26767.738676; stLENS1_750[751].fLow := 5.342722; stLENS1_750[751].fHigh := 13.396934; 
    stLENS1_750[752].fEnergy := 26821.327725; stLENS1_750[752].fLow := 5.323027; stLENS1_750[752].fHigh := 13.338777; 
    stLENS1_750[753].fEnergy := 26875.024059; stLENS1_750[753].fLow := 5.303404; stLENS1_750[753].fHigh := 13.280896; 
    stLENS1_750[754].fEnergy := 26928.827893; stLENS1_750[754].fLow := 5.283852; stLENS1_750[754].fHigh := 13.223288; 
    stLENS1_750[755].fEnergy := 26982.739442; stLENS1_750[755].fLow := 5.264371; stLENS1_750[755].fHigh := 13.165954; 
    stLENS1_750[756].fEnergy := 27036.758923; stLENS1_750[756].fLow := 5.244962; stLENS1_750[756].fHigh := 13.108890; 
    stLENS1_750[757].fEnergy := 27090.886550; stLENS1_750[757].fLow := 5.225623; stLENS1_750[757].fHigh := 13.052096; 
    stLENS1_750[758].fEnergy := 27145.122541; stLENS1_750[758].fLow := 5.206354; stLENS1_750[758].fHigh := 12.995570; 
    stLENS1_750[759].fEnergy := 27199.467113; stLENS1_750[759].fLow := 5.187155; stLENS1_750[759].fHigh := 12.939312; 
    stLENS1_750[760].fEnergy := 27253.920482; stLENS1_750[760].fLow := 5.168027; stLENS1_750[760].fHigh := 12.883319; 
    stLENS1_750[761].fEnergy := 27308.482867; stLENS1_750[761].fLow := 5.148968; stLENS1_750[761].fHigh := 12.827591; 
    stLENS1_750[762].fEnergy := 27363.154486; stLENS1_750[762].fLow := 5.129978; stLENS1_750[762].fHigh := 12.772126; 
    stLENS1_750[763].fEnergy := 27417.935558; stLENS1_750[763].fLow := 5.111057; stLENS1_750[763].fHigh := 12.716923; 
    stLENS1_750[764].fEnergy := 27472.826302; stLENS1_750[764].fLow := 5.092206; stLENS1_750[764].fHigh := 12.661979; 
    stLENS1_750[765].fEnergy := 27527.826937; stLENS1_750[765].fLow := 5.073423; stLENS1_750[765].fHigh := 12.607295; 
    stLENS1_750[766].fEnergy := 27582.937683; stLENS1_750[766].fLow := 5.054708; stLENS1_750[766].fHigh := 12.552869; 
    stLENS1_750[767].fEnergy := 27638.158761; stLENS1_750[767].fLow := 5.036062; stLENS1_750[767].fHigh := 12.498700; 
    stLENS1_750[768].fEnergy := 27693.490392; stLENS1_750[768].fLow := 5.017483; stLENS1_750[768].fHigh := 12.444785; 
    stLENS1_750[769].fEnergy := 27748.932796; stLENS1_750[769].fLow := 4.998973; stLENS1_750[769].fHigh := 12.391124; 
    stLENS1_750[770].fEnergy := 27804.486197; stLENS1_750[770].fLow := 4.980529; stLENS1_750[770].fHigh := 12.337716; 
    stLENS1_750[771].fEnergy := 27860.150815; stLENS1_750[771].fLow := 4.962153; stLENS1_750[771].fHigh := 12.284560; 
    stLENS1_750[772].fEnergy := 27915.926874; stLENS1_750[772].fLow := 4.943844; stLENS1_750[772].fHigh := 12.231653; 
    stLENS1_750[773].fEnergy := 27971.814597; stLENS1_750[773].fLow := 4.925601; stLENS1_750[773].fHigh := 12.178995; 
    stLENS1_750[774].fEnergy := 28027.814207; stLENS1_750[774].fLow := 4.907425; stLENS1_750[774].fHigh := 12.126585; 
    stLENS1_750[775].fEnergy := 28083.925929; stLENS1_750[775].fLow := 4.889315; stLENS1_750[775].fHigh := 12.074421; 
    stLENS1_750[776].fEnergy := 28140.149986; stLENS1_750[776].fLow := 4.871271; stLENS1_750[776].fHigh := 12.022503; 
    stLENS1_750[777].fEnergy := 28196.486604; stLENS1_750[777].fLow := 4.853293; stLENS1_750[777].fHigh := 11.970828; 
    stLENS1_750[778].fEnergy := 28252.936008; stLENS1_750[778].fLow := 4.835380; stLENS1_750[778].fHigh := 11.919396; 
    stLENS1_750[779].fEnergy := 28309.498423; stLENS1_750[779].fLow := 4.817533; stLENS1_750[779].fHigh := 11.868205; 
    stLENS1_750[780].fEnergy := 28366.174077; stLENS1_750[780].fLow := 4.799751; stLENS1_750[780].fHigh := 11.817254; 
    stLENS1_750[781].fEnergy := 28422.963195; stLENS1_750[781].fLow := 4.782033; stLENS1_750[781].fHigh := 11.766542; 
    stLENS1_750[782].fEnergy := 28479.866005; stLENS1_750[782].fLow := 4.764380; stLENS1_750[782].fHigh := 11.716069; 
    stLENS1_750[783].fEnergy := 28536.882735; stLENS1_750[783].fLow := 4.746791; stLENS1_750[783].fHigh := 11.665831; 
    stLENS1_750[784].fEnergy := 28594.013612; stLENS1_750[784].fLow := 4.729267; stLENS1_750[784].fHigh := 11.615829; 
    stLENS1_750[785].fEnergy := 28651.258866; stLENS1_750[785].fLow := 4.711806; stLENS1_750[785].fHigh := 11.566062; 
    stLENS1_750[786].fEnergy := 28708.618724; stLENS1_750[786].fLow := 4.694409; stLENS1_750[786].fHigh := 11.516527; 
    stLENS1_750[787].fEnergy := 28766.093417; stLENS1_750[787].fLow := 4.677076; stLENS1_750[787].fHigh := 11.467225; 
    stLENS1_750[788].fEnergy := 28823.683175; stLENS1_750[788].fLow := 4.659805; stLENS1_750[788].fHigh := 11.418153; 
    stLENS1_750[789].fEnergy := 28881.388227; stLENS1_750[789].fLow := 4.642598; stLENS1_750[789].fHigh := 11.369310; 
    stLENS1_750[790].fEnergy := 28939.208804; stLENS1_750[790].fLow := 4.625453; stLENS1_750[790].fHigh := 11.320696; 
    stLENS1_750[791].fEnergy := 28997.145139; stLENS1_750[791].fLow := 4.608371; stLENS1_750[791].fHigh := 11.272310; 
    stLENS1_750[792].fEnergy := 29055.197462; stLENS1_750[792].fLow := 4.591351; stLENS1_750[792].fHigh := 11.224149; 
    stLENS1_750[793].fEnergy := 29113.366006; stLENS1_750[793].fLow := 4.574393; stLENS1_750[793].fHigh := 11.176214; 
    stLENS1_750[794].fEnergy := 29171.651004; stLENS1_750[794].fLow := 4.557497; stLENS1_750[794].fHigh := 11.128502; 
    stLENS1_750[795].fEnergy := 29230.052688; stLENS1_750[795].fLow := 4.540663; stLENS1_750[795].fHigh := 11.081013; 
    stLENS1_750[796].fEnergy := 29288.571293; stLENS1_750[796].fLow := 4.523890; stLENS1_750[796].fHigh := 11.033746; 
    stLENS1_750[797].fEnergy := 29347.207052; stLENS1_750[797].fLow := 4.507178; stLENS1_750[797].fHigh := 10.986699; 
    stLENS1_750[798].fEnergy := 29405.960199; stLENS1_750[798].fLow := 4.490527; stLENS1_750[798].fHigh := 10.939872; 
    stLENS1_750[799].fEnergy := 29464.830971; stLENS1_750[799].fLow := 4.473937; stLENS1_750[799].fHigh := 10.893263; 
    stLENS1_750[800].fEnergy := 29523.819602; stLENS1_750[800].fLow := 4.457408; stLENS1_750[800].fHigh := 10.846872; 
    stLENS1_750[801].fEnergy := 29582.926328; stLENS1_750[801].fLow := 4.440938; stLENS1_750[801].fHigh := 10.800696; 
    stLENS1_750[802].fEnergy := 29642.151386; stLENS1_750[802].fLow := 4.424529; stLENS1_750[802].fHigh := 10.754736; 
    stLENS1_750[803].fEnergy := 29701.495012; stLENS1_750[803].fLow := 4.408180; stLENS1_750[803].fHigh := 10.708989; 
    stLENS1_750[804].fEnergy := 29760.957445; stLENS1_750[804].fLow := 4.391890; stLENS1_750[804].fHigh := 10.663456; 
    stLENS1_750[805].fEnergy := 29820.538922; stLENS1_750[805].fLow := 4.375660; stLENS1_750[805].fHigh := 10.618134; 
    stLENS1_750[806].fEnergy := 29880.239680; stLENS1_750[806].fLow := 4.359489; stLENS1_750[806].fHigh := 10.573024; 
    stLENS1_750[807].fEnergy := 29940.059960; stLENS1_750[807].fLow := 4.343377; stLENS1_750[807].fHigh := 10.528123; 
    stLENS1_750[808].fEnergy := 30000.000000; stLENS1_750[808].fLow := 4.327323; stLENS1_750[808].fHigh := 10.483431; 
    stLENS1_750[809].fEnergy := 30068.760232; stLENS1_750[809].fLow := 4.309031; stLENS1_750[809].fHigh := 10.432237; 
    stLENS1_750[810].fEnergy := 30128.957930; stLENS1_750[810].fLow := 4.293109; stLENS1_750[810].fHigh := 10.387863; 
    stLENS1_750[811].fEnergy := 30189.276144; stLENS1_750[811].fLow := 4.277245; stLENS1_750[811].fHigh := 10.343677; 
    stLENS1_750[812].fEnergy := 30249.715115; stLENS1_750[812].fLow := 4.261440; stLENS1_750[812].fHigh := 10.299679; 
    stLENS1_750[813].fEnergy := 30310.275085; stLENS1_750[813].fLow := 4.245693; stLENS1_750[813].fHigh := 10.255868; 
    stLENS1_750[814].fEnergy := 30370.956297; stLENS1_750[814].fLow := 4.230005; stLENS1_750[814].fHigh := 10.212244; 
    stLENS1_750[815].fEnergy := 30431.758992; stLENS1_750[815].fLow := 4.214374; stLENS1_750[815].fHigh := 10.168805; 
    stLENS1_750[816].fEnergy := 30492.683414; stLENS1_750[816].fLow := 4.198801; stLENS1_750[816].fHigh := 10.125551; 
    stLENS1_750[817].fEnergy := 30553.729807; stLENS1_750[817].fLow := 4.183286; stLENS1_750[817].fHigh := 10.082481; 
    stLENS1_750[818].fEnergy := 30614.898414; stLENS1_750[818].fLow := 4.167828; stLENS1_750[818].fHigh := 10.039594; 
    stLENS1_750[819].fEnergy := 30676.189482; stLENS1_750[819].fLow := 4.152427; stLENS1_750[819].fHigh := 9.996890; 
    stLENS1_750[820].fEnergy := 30737.603254; stLENS1_750[820].fLow := 4.137083; stLENS1_750[820].fHigh := 9.954367; 
    stLENS1_750[821].fEnergy := 30799.139977; stLENS1_750[821].fLow := 4.121796; stLENS1_750[821].fHigh := 9.912025; 
    stLENS1_750[822].fEnergy := 30860.799896; stLENS1_750[822].fLow := 4.106566; stLENS1_750[822].fHigh := 9.869863; 
    stLENS1_750[823].fEnergy := 30922.583259; stLENS1_750[823].fLow := 4.091391; stLENS1_750[823].fHigh := 9.827881; 
    stLENS1_750[824].fEnergy := 30984.490312; stLENS1_750[824].fLow := 4.076273; stLENS1_750[824].fHigh := 9.786077; 
    stLENS1_750[825].fEnergy := 31046.521303; stLENS1_750[825].fLow := 4.061210; stLENS1_750[825].fHigh := 9.744451; 
    stLENS1_750[826].fEnergy := 31108.676480; stLENS1_750[826].fLow := 4.046203; stLENS1_750[826].fHigh := 9.703002; 
    stLENS1_750[827].fEnergy := 31170.956091; stLENS1_750[827].fLow := 4.031252; stLENS1_750[827].fHigh := 9.661729; 
    stLENS1_750[828].fEnergy := 31233.360387; stLENS1_750[828].fLow := 4.016356; stLENS1_750[828].fHigh := 9.620632; 
    stLENS1_750[829].fEnergy := 31295.889616; stLENS1_750[829].fLow := 4.001515; stLENS1_750[829].fHigh := 9.579709; 
    stLENS1_750[830].fEnergy := 31358.544029; stLENS1_750[830].fLow := 3.986729; stLENS1_750[830].fHigh := 9.538961; 
    stLENS1_750[831].fEnergy := 31421.323876; stLENS1_750[831].fLow := 3.971997; stLENS1_750[831].fHigh := 9.498386; 
    stLENS1_750[832].fEnergy := 31484.229408; stLENS1_750[832].fLow := 3.957320; stLENS1_750[832].fHigh := 9.457984; 
    stLENS1_750[833].fEnergy := 31547.260878; stLENS1_750[833].fLow := 3.942697; stLENS1_750[833].fHigh := 9.417753; 
    stLENS1_750[834].fEnergy := 31610.418536; stLENS1_750[834].fLow := 3.928128; stLENS1_750[834].fHigh := 9.377694; 
